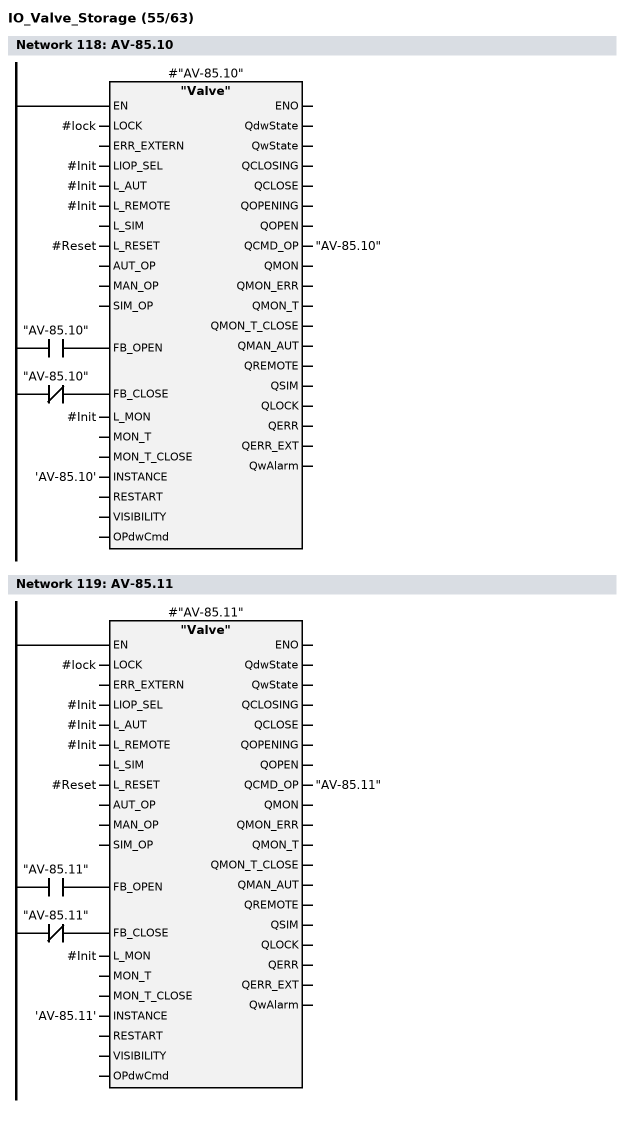
   RUNG wire#powerrail
      #"AV-85.10"(FB_OPEN := wire#w1, FB_CLOSE := wire#w2, LOCK := #lock, ERR_EXTERN :=, LIOP_SEL := #Init, L_AUT := #Init, L_REMOTE := #Init, L_SIM :=, L_RESET := #Reset, AUT_OP :=, MAN_OP :=, SIM_OP :=, L_MON := #Init, MON_T :=, MON_T_CLOSE :=, INSTANCE := 'AV-85.10', RESTART :=, VISIBILITY :=, OPdwCmd :=, QdwState =>, QwState =>, QCLOSING =>, QCLOSE =>, QOPENING =>, QOPEN =>, QCMD_OP => "AV-85.10", QMON =>, QMON_ERR =>, QMON_T =>, QMON_T_CLOSE =>, QMAN_AUT =>, QREMOTE =>, QSIM =>, QLOCK =>, QERR =>, QERR_EXT =>, QwAlarm =>)
   END_RUNG
   RUNG wire#powerrail
      Contact( "AV-85.10" )
   END_RUNG wire#w1
   RUNG wire#powerrail
      I_Contact( "AV-85.10" )
   END_RUNG wire#w2
   // the same network as SCL:
   #"AV-85.10"(LOCK := #lock,   // "Valve"
               LIOP_SEL := #Init,
               L_AUT := #Init,
               L_REMOTE := #Init,
               L_RESET := #Reset,
               FB_OPEN := "AV-85.10",
               FB_CLOSE := NOT "AV-85.10",
               L_MON := #Init,
               INSTANCE := 'AV-85.10',
               QCMD_OP => "AV-85.10");
END_REGION

REGION Network 119: AV-85.11
   RUNG wire#powerrail
      #"AV-85.11"(FB_OPEN := wire#w1, FB_CLOSE := wire#w2, LOCK := #lock, ERR_EXTERN :=, LIOP_SEL := #Init, L_AUT := #Init, L_REMOTE := #Init, L_SIM :=, L_RESET := #Reset, AUT_OP :=, MAN_OP :=, SIM_OP :=, L_MON := #Init, MON_T :=, MON_T_CLOSE :=, INSTANCE := 'AV-85.11', RESTART :=, VISIBILITY :=, OPdwCmd :=, QdwState =>, QwState =>, QCLOSING =>, QCLOSE =>, QOPENING =>, QOPEN =>, QCMD_OP => "AV-85.11", QMON =>, QMON_ERR =>, QMON_T =>, QMON_T_CLOSE =>, QMAN_AUT =>, QREMOTE =>, QSIM =>, QLOCK =>, QERR =>, QERR_EXT =>, QwAlarm =>)
   END_RUNG
   RUNG wire#powerrail
      Contact( "AV-85.11" )
   END_RUNG wire#w1
   RUNG wire#powerrail
      I_Contact( "AV-85.11" )
   END_RUNG wire#w2
   // the same network as SCL:
   #"AV-85.11"(LOCK := #lock,   // "Valve"
               LIOP_SEL := #Init,
               L_AUT := #Init,
               L_REMOTE := #Init,
               L_RESET := #Reset,
               FB_OPEN := "AV-85.11",
               FB_CLOSE := NOT "AV-85.11",
               L_MON := #Init,
               INSTANCE := 'AV-85.11',
               QCMD_OP => "AV-85.11");
END_REGION

REGION Network 120: AV-85.12
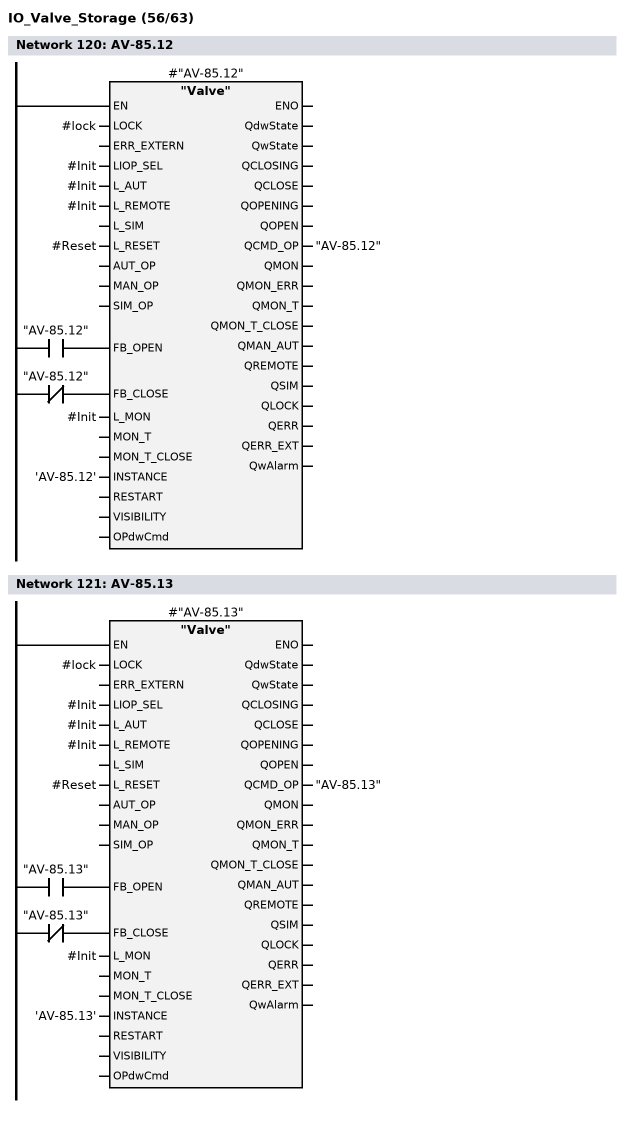
   RUNG wire#powerrail
      #"AV-85.12"(FB_OPEN := wire#w1, FB_CLOSE := wire#w2, LOCK := #lock, ERR_EXTERN :=, LIOP_SEL := #Init, L_AUT := #Init, L_REMOTE := #Init, L_SIM :=, L_RESET := #Reset, AUT_OP :=, MAN_OP :=, SIM_OP :=, L_MON := #Init, MON_T :=, MON_T_CLOSE :=, INSTANCE := 'AV-85.12', RESTART :=, VISIBILITY :=, OPdwCmd :=, QdwState =>, QwState =>, QCLOSING =>, QCLOSE =>, QOPENING =>, QOPEN =>, QCMD_OP => "AV-85.12", QMON =>, QMON_ERR =>, QMON_T =>, QMON_T_CLOSE =>, QMAN_AUT =>, QREMOTE =>, QSIM =>, QLOCK =>, QERR =>, QERR_EXT =>, QwAlarm =>)
   END_RUNG
   RUNG wire#powerrail
      Contact( "AV-85.12" )
   END_RUNG wire#w1
   RUNG wire#powerrail
      I_Contact( "AV-85.12" )
   END_RUNG wire#w2
   // the same network as SCL:
   #"AV-85.12"(LOCK := #lock,   // "Valve"
               LIOP_SEL := #Init,
               L_AUT := #Init,
               L_REMOTE := #Init,
               L_RESET := #Reset,
               FB_OPEN := "AV-85.12",
               FB_CLOSE := NOT "AV-85.12",
               L_MON := #Init,
               INSTANCE := 'AV-85.12',
               QCMD_OP => "AV-85.12");
END_REGION

REGION Network 121: AV-85.13
   RUNG wire#powerrail
      #"AV-85.13"(FB_OPEN := wire#w1, FB_CLOSE := wire#w2, LOCK := #lock, ERR_EXTERN :=, LIOP_SEL := #Init, L_AUT := #Init, L_REMOTE := #Init, L_SIM :=, L_RESET := #Reset, AUT_OP :=, MAN_OP :=, SIM_OP :=, L_MON := #Init, MON_T :=, MON_T_CLOSE :=, INSTANCE := 'AV-85.13', RESTART :=, VISIBILITY :=, OPdwCmd :=, QdwState =>, QwState =>, QCLOSING =>, QCLOSE =>, QOPENING =>, QOPEN =>, QCMD_OP => "AV-85.13", QMON =>, QMON_ERR =>, QMON_T =>, QMON_T_CLOSE =>, QMAN_AUT =>, QREMOTE =>, QSIM =>, QLOCK =>, QERR =>, QERR_EXT =>, QwAlarm =>)
   END_RUNG
   RUNG wire#powerrail
      Contact( "AV-85.13" )
   END_RUNG wire#w1
   RUNG wire#powerrail
      I_Contact( "AV-85.13" )
   END_RUNG wire#w2
   // the same network as SCL:
   #"AV-85.13"(LOCK := #lock,   // "Valve"
               LIOP_SEL := #Init,
               L_AUT := #Init,
               L_REMOTE := #Init,
               L_RESET := #Reset,
               FB_OPEN := "AV-85.13",
               FB_CLOSE := NOT "AV-85.13",
               L_MON := #Init,
               INSTANCE := 'AV-85.13',
               QCMD_OP => "AV-85.13");
END_REGION

REGION Network 122: AV-85.14
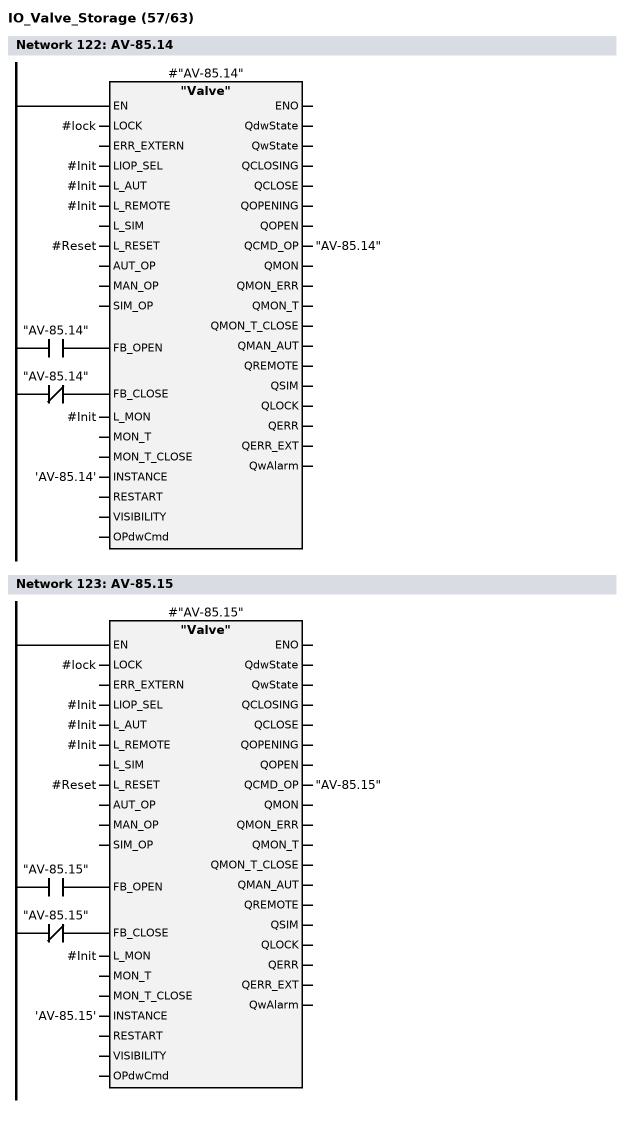
   RUNG wire#powerrail
      #"AV-85.14"(FB_OPEN := wire#w1, FB_CLOSE := wire#w2, LOCK := #lock, ERR_EXTERN :=, LIOP_SEL := #Init, L_AUT := #Init, L_REMOTE := #Init, L_SIM :=, L_RESET := #Reset, AUT_OP :=, MAN_OP :=, SIM_OP :=, L_MON := #Init, MON_T :=, MON_T_CLOSE :=, INSTANCE := 'AV-85.14', RESTART :=, VISIBILITY :=, OPdwCmd :=, QdwState =>, QwState =>, QCLOSING =>, QCLOSE =>, QOPENING =>, QOPEN =>, QCMD_OP => "AV-85.14", QMON =>, QMON_ERR =>, QMON_T =>, QMON_T_CLOSE =>, QMAN_AUT =>, QREMOTE =>, QSIM =>, QLOCK =>, QERR =>, QERR_EXT =>, QwAlarm =>)
   END_RUNG
   RUNG wire#powerrail
      Contact( "AV-85.14" )
   END_RUNG wire#w1
   RUNG wire#powerrail
      I_Contact( "AV-85.14" )
   END_RUNG wire#w2
   // the same network as SCL:
   #"AV-85.14"(LOCK := #lock,   // "Valve"
               LIOP_SEL := #Init,
               L_AUT := #Init,
               L_REMOTE := #Init,
               L_RESET := #Reset,
               FB_OPEN := "AV-85.14",
               FB_CLOSE := NOT "AV-85.14",
               L_MON := #Init,
               INSTANCE := 'AV-85.14',
               QCMD_OP => "AV-85.14");
END_REGION

REGION Network 123: AV-85.15
   RUNG wire#powerrail
      #"AV-85.15"(FB_OPEN := wire#w1, FB_CLOSE := wire#w2, LOCK := #lock, ERR_EXTERN :=, LIOP_SEL := #Init, L_AUT := #Init, L_REMOTE := #Init, L_SIM :=, L_RESET := #Reset, AUT_OP :=, MAN_OP :=, SIM_OP :=, L_MON := #Init, MON_T :=, MON_T_CLOSE :=, INSTANCE := 'AV-85.15', RESTART :=, VISIBILITY :=, OPdwCmd :=, QdwState =>, QwState =>, QCLOSING =>, QCLOSE =>, QOPENING =>, QOPEN =>, QCMD_OP => "AV-85.15", QMON =>, QMON_ERR =>, QMON_T =>, QMON_T_CLOSE =>, QMAN_AUT =>, QREMOTE =>, QSIM =>, QLOCK =>, QERR =>, QERR_EXT =>, QwAlarm =>)
   END_RUNG
   RUNG wire#powerrail
      Contact( "AV-85.15" )
   END_RUNG wire#w1
   RUNG wire#powerrail
      I_Contact( "AV-85.15" )
   END_RUNG wire#w2
   // the same network as SCL:
   #"AV-85.15"(LOCK := #lock,   // "Valve"
               LIOP_SEL := #Init,
               L_AUT := #Init,
               L_REMOTE := #Init,
               L_RESET := #Reset,
               FB_OPEN := "AV-85.15",
               FB_CLOSE := NOT "AV-85.15",
               L_MON := #Init,
               INSTANCE := 'AV-85.15',
               QCMD_OP => "AV-85.15");
END_REGION

REGION Network 124: AV-85.16
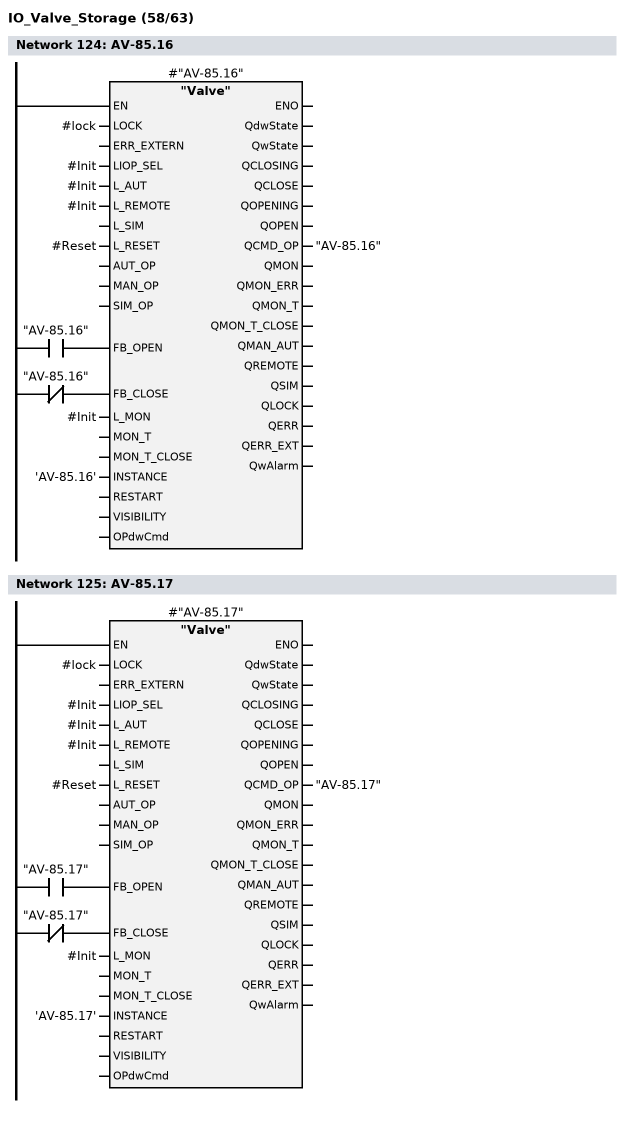
   RUNG wire#powerrail
      #"AV-85.16"(FB_OPEN := wire#w1, FB_CLOSE := wire#w2, LOCK := #lock, ERR_EXTERN :=, LIOP_SEL := #Init, L_AUT := #Init, L_REMOTE := #Init, L_SIM :=, L_RESET := #Reset, AUT_OP :=, MAN_OP :=, SIM_OP :=, L_MON := #Init, MON_T :=, MON_T_CLOSE :=, INSTANCE := 'AV-85.16', RESTART :=, VISIBILITY :=, OPdwCmd :=, QdwState =>, QwState =>, QCLOSING =>, QCLOSE =>, QOPENING =>, QOPEN =>, QCMD_OP => "AV-85.16", QMON =>, QMON_ERR =>, QMON_T =>, QMON_T_CLOSE =>, QMAN_AUT =>, QREMOTE =>, QSIM =>, QLOCK =>, QERR =>, QERR_EXT =>, QwAlarm =>)
   END_RUNG
   RUNG wire#powerrail
      Contact( "AV-85.16" )
   END_RUNG wire#w1
   RUNG wire#powerrail
      I_Contact( "AV-85.16" )
   END_RUNG wire#w2
   // the same network as SCL:
   #"AV-85.16"(LOCK := #lock,   // "Valve"
               LIOP_SEL := #Init,
               L_AUT := #Init,
               L_REMOTE := #Init,
               L_RESET := #Reset,
               FB_OPEN := "AV-85.16",
               FB_CLOSE := NOT "AV-85.16",
               L_MON := #Init,
               INSTANCE := 'AV-85.16',
               QCMD_OP => "AV-85.16");
END_REGION

REGION Network 125: AV-85.17
   RUNG wire#powerrail
      #"AV-85.17"(FB_OPEN := wire#w1, FB_CLOSE := wire#w2, LOCK := #lock, ERR_EXTERN :=, LIOP_SEL := #Init, L_AUT := #Init, L_REMOTE := #Init, L_SIM :=, L_RESET := #Reset, AUT_OP :=, MAN_OP :=, SIM_OP :=, L_MON := #Init, MON_T :=, MON_T_CLOSE :=, INSTANCE := 'AV-85.17', RESTART :=, VISIBILITY :=, OPdwCmd :=, QdwState =>, QwState =>, QCLOSING =>, QCLOSE =>, QOPENING =>, QOPEN =>, QCMD_OP => "AV-85.17", QMON =>, QMON_ERR =>, QMON_T =>, QMON_T_CLOSE =>, QMAN_AUT =>, QREMOTE =>, QSIM =>, QLOCK =>, QERR =>, QERR_EXT =>, QwAlarm =>)
   END_RUNG
   RUNG wire#powerrail
      Contact( "AV-85.17" )
   END_RUNG wire#w1
   RUNG wire#powerrail
      I_Contact( "AV-85.17" )
   END_RUNG wire#w2
   // the same network as SCL:
   #"AV-85.17"(LOCK := #lock,   // "Valve"
               LIOP_SEL := #Init,
               L_AUT := #Init,
               L_REMOTE := #Init,
               L_RESET := #Reset,
               FB_OPEN := "AV-85.17",
               FB_CLOSE := NOT "AV-85.17",
               L_MON := #Init,
               INSTANCE := 'AV-85.17',
               QCMD_OP => "AV-85.17");
END_REGION

REGION Network 126: AV-85.18
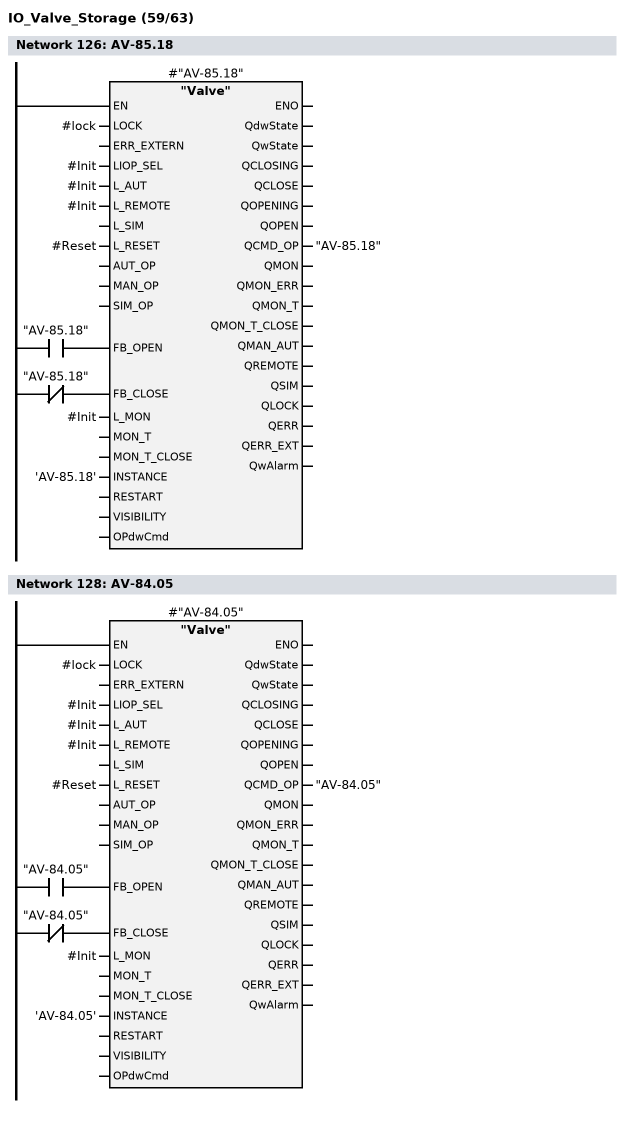
   RUNG wire#powerrail
      #"AV-85.18"(FB_OPEN := wire#w1, FB_CLOSE := wire#w2, LOCK := #lock, ERR_EXTERN :=, LIOP_SEL := #Init, L_AUT := #Init, L_REMOTE := #Init, L_SIM :=, L_RESET := #Reset, AUT_OP :=, MAN_OP :=, SIM_OP :=, L_MON := #Init, MON_T :=, MON_T_CLOSE :=, INSTANCE := 'AV-85.18', RESTART :=, VISIBILITY :=, OPdwCmd :=, QdwState =>, QwState =>, QCLOSING =>, QCLOSE =>, QOPENING =>, QOPEN =>, QCMD_OP => "AV-85.18", QMON =>, QMON_ERR =>, QMON_T =>, QMON_T_CLOSE =>, QMAN_AUT =>, QREMOTE =>, QSIM =>, QLOCK =>, QERR =>, QERR_EXT =>, QwAlarm =>)
   END_RUNG
   RUNG wire#powerrail
      Contact( "AV-85.18" )
   END_RUNG wire#w1
   RUNG wire#powerrail
      I_Contact( "AV-85.18" )
   END_RUNG wire#w2
   // the same network as SCL:
   #"AV-85.18"(LOCK := #lock,   // "Valve"
               LIOP_SEL := #Init,
               L_AUT := #Init,
               L_REMOTE := #Init,
               L_RESET := #Reset,
               FB_OPEN := "AV-85.18",
               FB_CLOSE := NOT "AV-85.18",
               L_MON := #Init,
               INSTANCE := 'AV-85.18',
               QCMD_OP => "AV-85.18");
END_REGION

REGION Network 128: AV-84.05
   RUNG wire#powerrail
      #"AV-84.05"(FB_OPEN := wire#w1, FB_CLOSE := wire#w2, LOCK := #lock, ERR_EXTERN :=, LIOP_SEL := #Init, L_AUT := #Init, L_REMOTE := #Init, L_SIM :=, L_RESET := #Reset, AUT_OP :=, MAN_OP :=, SIM_OP :=, L_MON := #Init, MON_T :=, MON_T_CLOSE :=, INSTANCE := 'AV-84.05', RESTART :=, VISIBILITY :=, OPdwCmd :=, QdwState =>, QwState =>, QCLOSING =>, QCLOSE =>, QOPENING =>, QOPEN =>, QCMD_OP => "AV-84.05", QMON =>, QMON_ERR =>, QMON_T =>, QMON_T_CLOSE =>, QMAN_AUT =>, QREMOTE =>, QSIM =>, QLOCK =>, QERR =>, QERR_EXT =>, QwAlarm =>)
   END_RUNG
   RUNG wire#powerrail
      Contact( "AV-84.05" )
   END_RUNG wire#w1
   RUNG wire#powerrail
      I_Contact( "AV-84.05" )
   END_RUNG wire#w2
   // the same network as SCL:
   #"AV-84.05"(LOCK := #lock,   // "Valve"
               LIOP_SEL := #Init,
               L_AUT := #Init,
               L_REMOTE := #Init,
               L_RESET := #Reset,
               FB_OPEN := "AV-84.05",
               FB_CLOSE := NOT "AV-84.05",
               L_MON := #Init,
               INSTANCE := 'AV-84.05',
               QCMD_OP => "AV-84.05");
END_REGION

REGION Network 129: AV-84.06
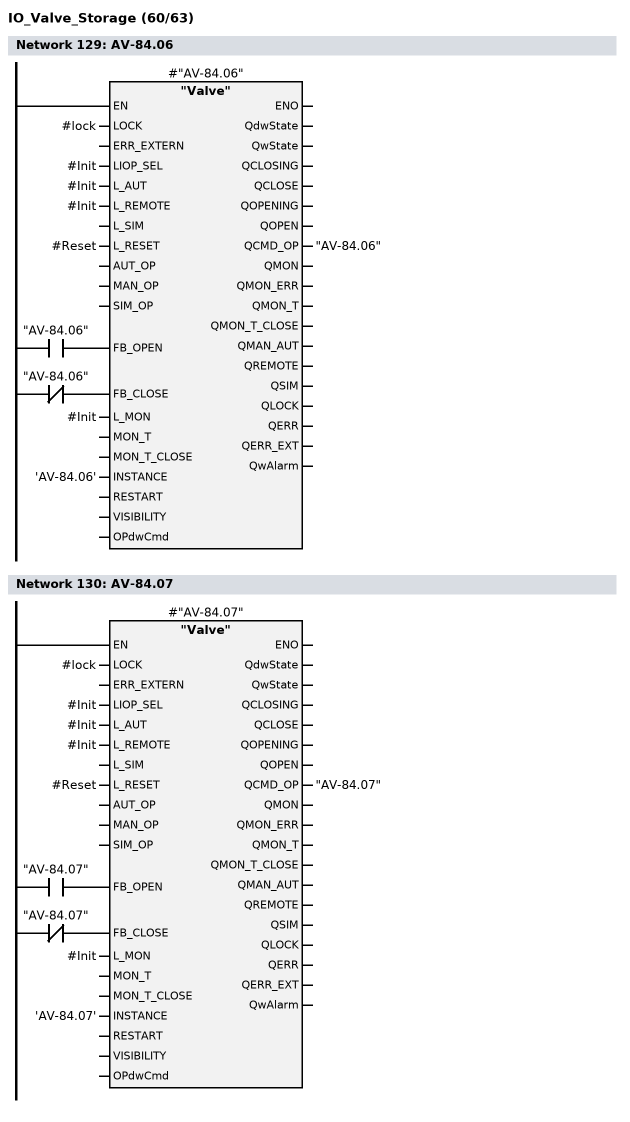
   RUNG wire#powerrail
      #"AV-84.06"(FB_OPEN := wire#w1, FB_CLOSE := wire#w2, LOCK := #lock, ERR_EXTERN :=, LIOP_SEL := #Init, L_AUT := #Init, L_REMOTE := #Init, L_SIM :=, L_RESET := #Reset, AUT_OP :=, MAN_OP :=, SIM_OP :=, L_MON := #Init, MON_T :=, MON_T_CLOSE :=, INSTANCE := 'AV-84.06', RESTART :=, VISIBILITY :=, OPdwCmd :=, QdwState =>, QwState =>, QCLOSING =>, QCLOSE =>, QOPENING =>, QOPEN =>, QCMD_OP => "AV-84.06", QMON =>, QMON_ERR =>, QMON_T =>, QMON_T_CLOSE =>, QMAN_AUT =>, QREMOTE =>, QSIM =>, QLOCK =>, QERR =>, QERR_EXT =>, QwAlarm =>)
   END_RUNG
   RUNG wire#powerrail
      Contact( "AV-84.06" )
   END_RUNG wire#w1
   RUNG wire#powerrail
      I_Contact( "AV-84.06" )
   END_RUNG wire#w2
   // the same network as SCL:
   #"AV-84.06"(LOCK := #lock,   // "Valve"
               LIOP_SEL := #Init,
               L_AUT := #Init,
               L_REMOTE := #Init,
               L_RESET := #Reset,
               FB_OPEN := "AV-84.06",
               FB_CLOSE := NOT "AV-84.06",
               L_MON := #Init,
               INSTANCE := 'AV-84.06',
               QCMD_OP => "AV-84.06");
END_REGION

REGION Network 130: AV-84.07
   RUNG wire#powerrail
      #"AV-84.07"(FB_OPEN := wire#w1, FB_CLOSE := wire#w2, LOCK := #lock, ERR_EXTERN :=, LIOP_SEL := #Init, L_AUT := #Init, L_REMOTE := #Init, L_SIM :=, L_RESET := #Reset, AUT_OP :=, MAN_OP :=, SIM_OP :=, L_MON := #Init, MON_T :=, MON_T_CLOSE :=, INSTANCE := 'AV-84.07', RESTART :=, VISIBILITY :=, OPdwCmd :=, QdwState =>, QwState =>, QCLOSING =>, QCLOSE =>, QOPENING =>, QOPEN =>, QCMD_OP => "AV-84.07", QMON =>, QMON_ERR =>, QMON_T =>, QMON_T_CLOSE =>, QMAN_AUT =>, QREMOTE =>, QSIM =>, QLOCK =>, QERR =>, QERR_EXT =>, QwAlarm =>)
   END_RUNG
   RUNG wire#powerrail
      Contact( "AV-84.07" )
   END_RUNG wire#w1
   RUNG wire#powerrail
      I_Contact( "AV-84.07" )
   END_RUNG wire#w2
   // the same network as SCL:
   #"AV-84.07"(LOCK := #lock,   // "Valve"
               LIOP_SEL := #Init,
               L_AUT := #Init,
               L_REMOTE := #Init,
               L_RESET := #Reset,
               FB_OPEN := "AV-84.07",
               FB_CLOSE := NOT "AV-84.07",
               L_MON := #Init,
               INSTANCE := 'AV-84.07',
               QCMD_OP => "AV-84.07");
END_REGION

REGION Network 131: AV-84.08
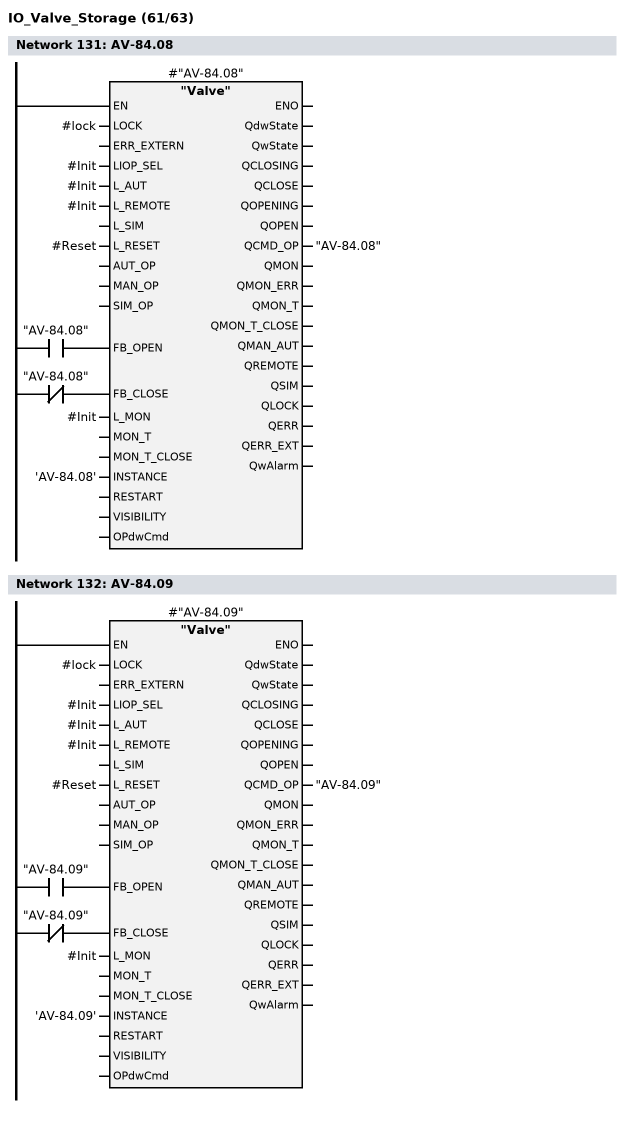
   RUNG wire#powerrail
      #"AV-84.08"(FB_OPEN := wire#w1, FB_CLOSE := wire#w2, LOCK := #lock, ERR_EXTERN :=, LIOP_SEL := #Init, L_AUT := #Init, L_REMOTE := #Init, L_SIM :=, L_RESET := #Reset, AUT_OP :=, MAN_OP :=, SIM_OP :=, L_MON := #Init, MON_T :=, MON_T_CLOSE :=, INSTANCE := 'AV-84.08', RESTART :=, VISIBILITY :=, OPdwCmd :=, QdwState =>, QwState =>, QCLOSING =>, QCLOSE =>, QOPENING =>, QOPEN =>, QCMD_OP => "AV-84.08", QMON =>, QMON_ERR =>, QMON_T =>, QMON_T_CLOSE =>, QMAN_AUT =>, QREMOTE =>, QSIM =>, QLOCK =>, QERR =>, QERR_EXT =>, QwAlarm =>)
   END_RUNG
   RUNG wire#powerrail
      Contact( "AV-84.08" )
   END_RUNG wire#w1
   RUNG wire#powerrail
      I_Contact( "AV-84.08" )
   END_RUNG wire#w2
   // the same network as SCL:
   #"AV-84.08"(LOCK := #lock,   // "Valve"
               LIOP_SEL := #Init,
               L_AUT := #Init,
               L_REMOTE := #Init,
               L_RESET := #Reset,
               FB_OPEN := "AV-84.08",
               FB_CLOSE := NOT "AV-84.08",
               L_MON := #Init,
               INSTANCE := 'AV-84.08',
               QCMD_OP => "AV-84.08");
END_REGION

REGION Network 132: AV-84.09
   RUNG wire#powerrail
      #"AV-84.09"(FB_OPEN := wire#w1, FB_CLOSE := wire#w2, LOCK := #lock, ERR_EXTERN :=, LIOP_SEL := #Init, L_AUT := #Init, L_REMOTE := #Init, L_SIM :=, L_RESET := #Reset, AUT_OP :=, MAN_OP :=, SIM_OP :=, L_MON := #Init, MON_T :=, MON_T_CLOSE :=, INSTANCE := 'AV-84.09', RESTART :=, VISIBILITY :=, OPdwCmd :=, QdwState =>, QwState =>, QCLOSING =>, QCLOSE =>, QOPENING =>, QOPEN =>, QCMD_OP => "AV-84.09", QMON =>, QMON_ERR =>, QMON_T =>, QMON_T_CLOSE =>, QMAN_AUT =>, QREMOTE =>, QSIM =>, QLOCK =>, QERR =>, QERR_EXT =>, QwAlarm =>)
   END_RUNG
   RUNG wire#powerrail
      Contact( "AV-84.09" )
   END_RUNG wire#w1
   RUNG wire#powerrail
      I_Contact( "AV-84.09" )
   END_RUNG wire#w2
   // the same network as SCL:
   #"AV-84.09"(LOCK := #lock,   // "Valve"
               LIOP_SEL := #Init,
               L_AUT := #Init,
               L_REMOTE := #Init,
               L_RESET := #Reset,
               FB_OPEN := "AV-84.09",
               FB_CLOSE := NOT "AV-84.09",
               L_MON := #Init,
               INSTANCE := 'AV-84.09',
               QCMD_OP => "AV-84.09");
END_REGION

REGION Network 133: AV-84.10
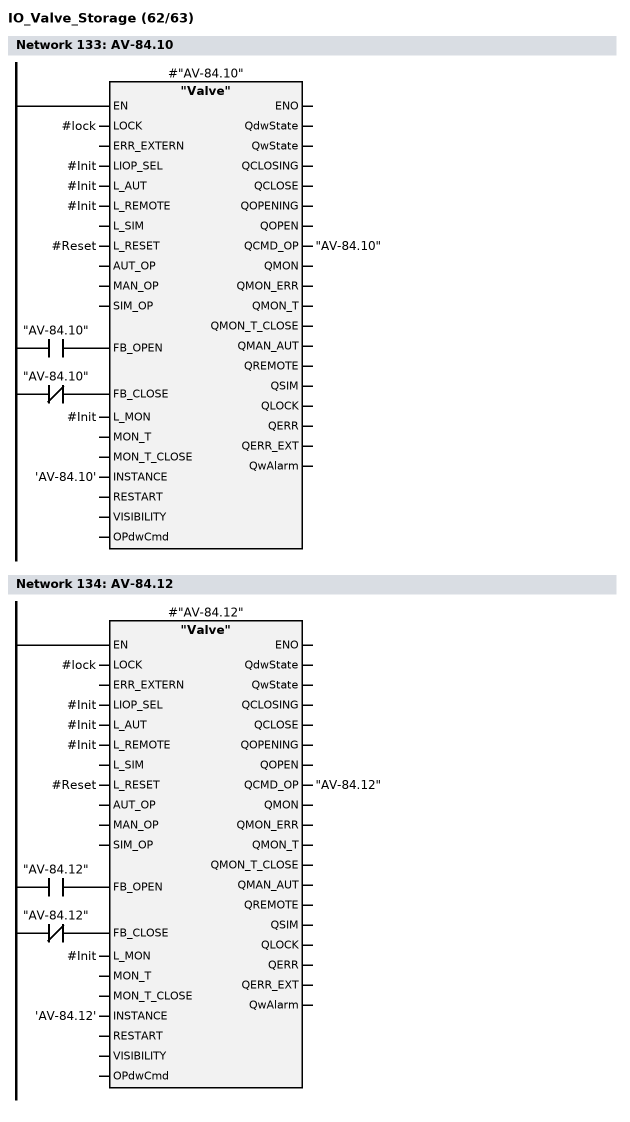
   RUNG wire#powerrail
      #"AV-84.10"(FB_OPEN := wire#w1, FB_CLOSE := wire#w2, LOCK := #lock, ERR_EXTERN :=, LIOP_SEL := #Init, L_AUT := #Init, L_REMOTE := #Init, L_SIM :=, L_RESET := #Reset, AUT_OP :=, MAN_OP :=, SIM_OP :=, L_MON := #Init, MON_T :=, MON_T_CLOSE :=, INSTANCE := 'AV-84.10', RESTART :=, VISIBILITY :=, OPdwCmd :=, QdwState =>, QwState =>, QCLOSING =>, QCLOSE =>, QOPENING =>, QOPEN =>, QCMD_OP => "AV-84.10", QMON =>, QMON_ERR =>, QMON_T =>, QMON_T_CLOSE =>, QMAN_AUT =>, QREMOTE =>, QSIM =>, QLOCK =>, QERR =>, QERR_EXT =>, QwAlarm =>)
   END_RUNG
   RUNG wire#powerrail
      Contact( "AV-84.10" )
   END_RUNG wire#w1
   RUNG wire#powerrail
      I_Contact( "AV-84.10" )
   END_RUNG wire#w2
   // the same network as SCL:
   #"AV-84.10"(LOCK := #lock,   // "Valve"
               LIOP_SEL := #Init,
               L_AUT := #Init,
               L_REMOTE := #Init,
               L_RESET := #Reset,
               FB_OPEN := "AV-84.10",
               FB_CLOSE := NOT "AV-84.10",
               L_MON := #Init,
               INSTANCE := 'AV-84.10',
               QCMD_OP => "AV-84.10");
END_REGION

REGION Network 134: AV-84.12
   RUNG wire#powerrail
      #"AV-84.12"(FB_OPEN := wire#w1, FB_CLOSE := wire#w2, LOCK := #lock, ERR_EXTERN :=, LIOP_SEL := #Init, L_AUT := #Init, L_REMOTE := #Init, L_SIM :=, L_RESET := #Reset, AUT_OP :=, MAN_OP :=, SIM_OP :=, L_MON := #Init, MON_T :=, MON_T_CLOSE :=, INSTANCE := 'AV-84.12', RESTART :=, VISIBILITY :=, OPdwCmd :=, QdwState =>, QwState =>, QCLOSING =>, QCLOSE =>, QOPENING =>, QOPEN =>, QCMD_OP => "AV-84.12", QMON =>, QMON_ERR =>, QMON_T =>, QMON_T_CLOSE =>, QMAN_AUT =>, QREMOTE =>, QSIM =>, QLOCK =>, QERR =>, QERR_EXT =>, QwAlarm =>)
   END_RUNG
   RUNG wire#powerrail
      Contact( "AV-84.12" )
   END_RUNG wire#w1
   RUNG wire#powerrail
      I_Contact( "AV-84.12" )
   END_RUNG wire#w2
   // the same network as SCL:
   #"AV-84.12"(LOCK := #lock,   // "Valve"
               LIOP_SEL := #Init,
               L_AUT := #Init,
               L_REMOTE := #Init,
               L_RESET := #Reset,
               FB_OPEN := "AV-84.12",
               FB_CLOSE := NOT "AV-84.12",
               L_MON := #Init,
               INSTANCE := 'AV-84.12',
               QCMD_OP => "AV-84.12");
END_REGION

REGION Network 135: AV-84.13
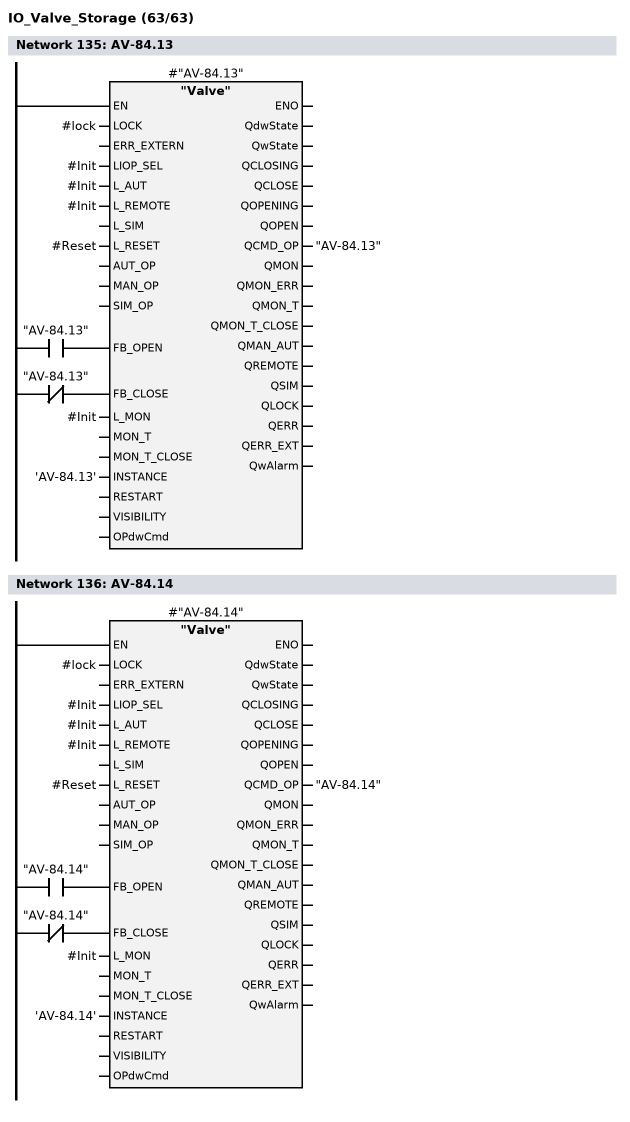
   RUNG wire#powerrail
      #"AV-84.13"(FB_OPEN := wire#w1, FB_CLOSE := wire#w2, LOCK := #lock, ERR_EXTERN :=, LIOP_SEL := #Init, L_AUT := #Init, L_REMOTE := #Init, L_SIM :=, L_RESET := #Reset, AUT_OP :=, MAN_OP :=, SIM_OP :=, L_MON := #Init, MON_T :=, MON_T_CLOSE :=, INSTANCE := 'AV-84.13', RESTART :=, VISIBILITY :=, OPdwCmd :=, QdwState =>, QwState =>, QCLOSING =>, QCLOSE =>, QOPENING =>, QOPEN =>, QCMD_OP => "AV-84.13", QMON =>, QMON_ERR =>, QMON_T =>, QMON_T_CLOSE =>, QMAN_AUT =>, QREMOTE =>, QSIM =>, QLOCK =>, QERR =>, QERR_EXT =>, QwAlarm =>)
   END_RUNG
   RUNG wire#powerrail
      Contact( "AV-84.13" )
   END_RUNG wire#w1
   RUNG wire#powerrail
      I_Contact( "AV-84.13" )
   END_RUNG wire#w2
   // the same network as SCL:
   #"AV-84.13"(LOCK := #lock,   // "Valve"
               LIOP_SEL := #Init,
               L_AUT := #Init,
               L_REMOTE := #Init,
               L_RESET := #Reset,
               FB_OPEN := "AV-84.13",
               FB_CLOSE := NOT "AV-84.13",
               L_MON := #Init,
               INSTANCE := 'AV-84.13',
               QCMD_OP => "AV-84.13");
END_REGION

REGION Network 136: AV-84.14
   RUNG wire#powerrail
      #"AV-84.14"(FB_OPEN := wire#w1, FB_CLOSE := wire#w2, LOCK := #lock, ERR_EXTERN :=, LIOP_SEL := #Init, L_AUT := #Init, L_REMOTE := #Init, L_SIM :=, L_RESET := #Reset, AUT_OP :=, MAN_OP :=, SIM_OP :=, L_MON := #Init, MON_T :=, MON_T_CLOSE :=, INSTANCE := 'AV-84.14', RESTART :=, VISIBILITY :=, OPdwCmd :=, QdwState =>, QwState =>, QCLOSING =>, QCLOSE =>, QOPENING =>, QOPEN =>, QCMD_OP => "AV-84.14", QMON =>, QMON_ERR =>, QMON_T =>, QMON_T_CLOSE =>, QMAN_AUT =>, QREMOTE =>, QSIM =>, QLOCK =>, QERR =>, QERR_EXT =>, QwAlarm =>)
   END_RUNG
   RUNG wire#powerrail
      Contact( "AV-84.14" )
   END_RUNG wire#w1
   RUNG wire#powerrail
      I_Contact( "AV-84.14" )
   END_RUNG wire#w2
   // the same network as SCL:
   #"AV-84.14"(LOCK := #lock,   // "Valve"
               LIOP_SEL := #Init,
               L_AUT := #Init,
               L_REMOTE := #Init,
               L_RESET := #Reset,
               FB_OPEN := "AV-84.14",
               FB_CLOSE := NOT "AV-84.14",
               L_MON := #Init,
               INSTANCE := 'AV-84.14',
               QCMD_OP => "AV-84.14");
END_REGION
END_FUNCTION_BLOCK

FUNCTION_BLOCK "IO_Digital_Storage"   // FB22, LAD
{ S7_Optimized_Access := 'TRUE' }
VERSION : 0.1
// stored: AutoNumber false, IsIECCheckEnabled false, IsRetainMemResEnabled false, MemoryReserve 100, SetENOAutomatically false, UDAEnableTagReadback false
   VAR_INPUT
      lock : Bool;
      init : Bool;
      Reset : Bool;
   END_VAR
   VAR
      "FS-23.01" : "Digital";
      "FS-24.01" { S7_SetPoint := 'True'} : "Digital";
      "FS-34.01" { S7_SetPoint := 'True'} : "Digital";
      "FS-35.01" { S7_SetPoint := 'True'} : "Digital";
   END_VAR
BEGIN

REGION Network 1: FS-23.01
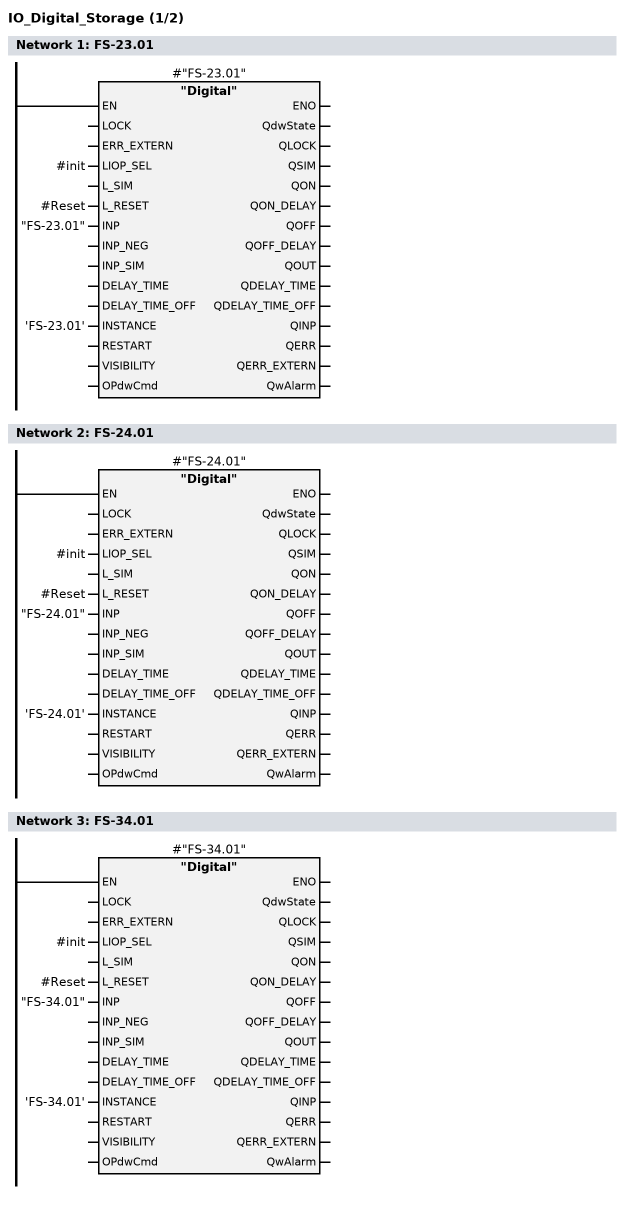
   RUNG wire#powerrail
      #"FS-23.01"(LOCK :=, ERR_EXTERN :=, LIOP_SEL := #init, L_SIM :=, L_RESET := #Reset, INP := "FS-23.01", INP_NEG :=, INP_SIM :=, DELAY_TIME :=, DELAY_TIME_OFF :=, INSTANCE := 'FS-23.01', RESTART :=, VISIBILITY :=, OPdwCmd :=, QdwState =>, QLOCK =>, QSIM =>, QON =>, QON_DELAY =>, QOFF =>, QOFF_DELAY =>, QOUT =>, QDELAY_TIME =>, QDELAY_TIME_OFF =>, QINP =>, QERR =>, QERR_EXTERN =>, QwAlarm =>)
   END_RUNG
   // the same network as SCL:
   #"FS-23.01"(LIOP_SEL := #init, L_RESET := #Reset, INP := "FS-23.01", INSTANCE := 'FS-23.01');   // "Digital"
END_REGION

REGION Network 2: FS-24.01
   RUNG wire#powerrail
      #"FS-24.01"(LOCK :=, ERR_EXTERN :=, LIOP_SEL := #init, L_SIM :=, L_RESET := #Reset, INP := "FS-24.01", INP_NEG :=, INP_SIM :=, DELAY_TIME :=, DELAY_TIME_OFF :=, INSTANCE := 'FS-24.01', RESTART :=, VISIBILITY :=, OPdwCmd :=, QdwState =>, QLOCK =>, QSIM =>, QON =>, QON_DELAY =>, QOFF =>, QOFF_DELAY =>, QOUT =>, QDELAY_TIME =>, QDELAY_TIME_OFF =>, QINP =>, QERR =>, QERR_EXTERN =>, QwAlarm =>)
   END_RUNG
   // the same network as SCL:
   #"FS-24.01"(LIOP_SEL := #init, L_RESET := #Reset, INP := "FS-24.01", INSTANCE := 'FS-24.01');   // "Digital"
END_REGION

REGION Network 3: FS-34.01
   RUNG wire#powerrail
      #"FS-34.01"(LOCK :=, ERR_EXTERN :=, LIOP_SEL := #init, L_SIM :=, L_RESET := #Reset, INP := "FS-34.01", INP_NEG :=, INP_SIM :=, DELAY_TIME :=, DELAY_TIME_OFF :=, INSTANCE := 'FS-34.01', RESTART :=, VISIBILITY :=, OPdwCmd :=, QdwState =>, QLOCK =>, QSIM =>, QON =>, QON_DELAY =>, QOFF =>, QOFF_DELAY =>, QOUT =>, QDELAY_TIME =>, QDELAY_TIME_OFF =>, QINP =>, QERR =>, QERR_EXTERN =>, QwAlarm =>)
   END_RUNG
   // the same network as SCL:
   #"FS-34.01"(LIOP_SEL := #init, L_RESET := #Reset, INP := "FS-34.01", INSTANCE := 'FS-34.01');   // "Digital"
END_REGION

REGION Network 4: FS-35.01
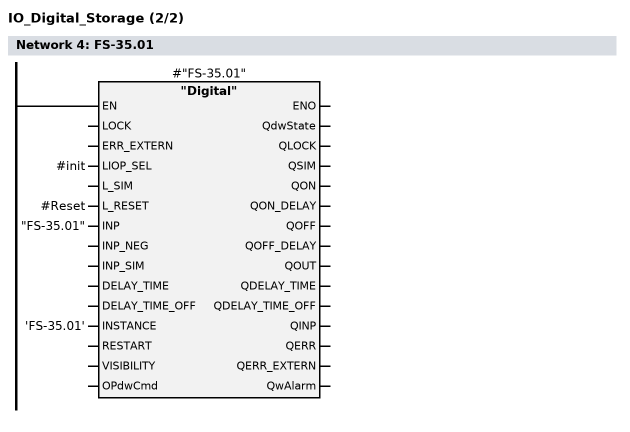
   RUNG wire#powerrail
      #"FS-35.01"(LOCK :=, ERR_EXTERN :=, LIOP_SEL := #init, L_SIM :=, L_RESET := #Reset, INP := "FS-35.01", INP_NEG :=, INP_SIM :=, DELAY_TIME :=, DELAY_TIME_OFF :=, INSTANCE := 'FS-35.01', RESTART :=, VISIBILITY :=, OPdwCmd :=, QdwState =>, QLOCK =>, QSIM =>, QON =>, QON_DELAY =>, QOFF =>, QOFF_DELAY =>, QOUT =>, QDELAY_TIME =>, QDELAY_TIME_OFF =>, QINP =>, QERR =>, QERR_EXTERN =>, QwAlarm =>)
   END_RUNG
   // the same network as SCL:
   #"FS-35.01"(LIOP_SEL := #init, L_RESET := #Reset, INP := "FS-35.01", INSTANCE := 'FS-35.01');   // "Digital"
END_REGION
END_FUNCTION_BLOCK

FUNCTION_BLOCK "Storage_Tank_Single_Inload"   // FB21, LAD
{ S7_Optimized_Access := 'FALSE' }
VERSION : 0.1
// stored: AutoNumber true, IsIECCheckEnabled false, SetENOAutomatically false, UDAEnableTagReadback false
   VAR_INPUT
      Level_Bypass : Bool;
      Single_CIP_Cmd : Bool;
      IN_FBAV_Load : Bool;
      IN_FBAV_Transfer : Bool;
      IN_FBP_Transfer : Bool;
      IN_FBP_Transfer_Speed : Real;
      IN_FBP_CIP : Bool;
      IN_FBAV_CIP_Sup : Bool;
      IN_FBAV_CIP_Tank : Bool;
      IN_FBAV_CIP_Line : Bool;
      IN_LT01 : Real;
      IN_FS : Bool;
      CIP_Req_OK : Bool;
      CIP_ON_Progress : Bool;
      CIP_Supply_ON : Bool;
      CIP_Complete : Bool;
      CIPPulse : Bool;
      Filler_Product_Req : Bool;
      Filler_CIP_Req : Bool;
      Loading_Busy : Bool;
      Transfer_Busy : Bool;
   END_VAR
   VAR_OUTPUT
      Out_AV_Load : Bool;
      Out_AV_Transfer : Bool;
      Out_P_Transfer : Bool;
      Out_P_TF_Speed : Real;
      Out_P_CIP : Bool;
      Out_AV_CIP_Line : Bool;
      Out_AV_CIP_Tank : Bool;
      Out_AV_CIP_Filling : Bool;
      CIP_Tank_Req : Bool;
      CIP_Line_Req : Bool;
      CIP_LineOK : Bool;
   END_VAR
   VAR DB_SPECIFIC
      Cmd : Struct
         Inload_Select_Tank : Bool;
         Inload : Bool;   // Start Loading
         Tank_CIP_Req : Bool;
         Line_CIP_Req : Bool;
         Tank_Filling_CIP_Req : Bool;
         CIP_Filling_En : Bool;
         CIP_Line_Req_OK : Bool;
         CIP_Supply_ON : Bool;
         CIP_ON_Progress : Bool;
         Flushing : Bool;   // Water Flushing
         RaadyForTF : Bool;   // Tank Ready for Blending
         Flush_Select : Byte;
         Drain_In : Bool;
         Drain_Transfer : Bool;
      END_STRUCT;
      Param : Struct
         SP_Level_LL : Real := 10.0;
         SP_Level_ML : Real := 80.0;
         SP_Level_HL : Real := 100.0;
         SupplyPump_SP_Speed : Real := 80.0;
         L_Hi_Lim : Real := 100.0;
         L_Lo_Lim : Real := 0.0;
         L_Hys : Real := 2.0;
         FlushingTime : DInt := 10000;
         CIP_Trf_SP_Speed : Real := 80.0;
         CIP_Ret_ON_SP : Real := 10.0;
         CIP_Ret_OFF_SP : Real;
         Transfer_P_Speed : Real := 60.0;
         Drain_Inload_SP : DInt := 10;
         Drain_Transfer_SP : DInt := 10;
      END_STRUCT;
      State : Struct   // Tank in loading state
         Tank_inloading : Bool;
         Tank_inCIP : Bool;
         Tank_Filling_inCIP : Bool;
         Line_inCIP : Bool;
         FIlling_inCIP : Bool;
         Flushing : Bool;
         Tank_LL : Bool;
         Tank_ML : Bool;
         Tank_HL : Bool;
         Inload_Enable : Bool;
         Tank_CIP_Enable : Bool;
         Line_CIP_Enable : Bool;
         Tank_Filling_CIP_Enable : Bool;
         Flushing_Enable : Bool;
         Flush_selected : Byte;
         CIP_Request_OK : Bool;
         CIP_ReturnON : Bool;
         Ready_For_Transfer_EN : Bool;   // Tank Ready for Transfer to Blending
         Ready_For_Transfer : Bool;   // Tank Ready for Transfer to Blending
         HWT_Status : Int;
         Transfer_to_Filling : Bool;
         "Line_AV4&AV5" : Bool;
         "Line_AV1&AV2" : Bool;
         "Line_AV7&AV8" : Bool;
         "Line_AV10&AV11" : Bool;
         "Line_AV5&AV6" : Bool;
         CIP_Line1_ON : Bool;
         CIP_Line2_ON : Bool;
         CIP_Line3_ON : Bool;
         CIP_Line4_ON : Bool;
         Drain_Inload : Bool;
         Drain_Transfer : Bool;
      END_STRUCT;
      alwaysON : Bool;
      L_Hys_Abs : Real;
      Hys_Level_HL : Real;
      Hys_Level_ML : Real;
      Hys_Level_LL : Real;
      Drain_Inload_MSec : DInt;
      Drain_Inload_Count : IEC_DCOUNTER;
      Drain_Inload_Act { S7_SetPoint := 'True'} : DInt;
      Drain_Transfer_MSec : DInt;
      Drain_Transfer_Count : IEC_DCOUNTER;
      Drain_Transfer_Act : DInt;
      r : Struct
         PosE1 : Bool;
         PosE2 : Bool;
         PosE3 : Bool;
         PosE4 : Bool;
         PosE5 : Bool;
         PosE6 : Bool;
         PosE7 : Bool;
         PosE8 : Bool;
         PosE9 : Bool;
         PosE10 : Bool;
         PosE11 : Bool;
         PosE12 : Bool;
         PosE13 : Bool;
         PosE14 : Bool;
         PosE15 : Bool;
         PosE16 : Bool;
         PosE17 : Bool;
         PosE18 : Bool;
         PosE19 : Bool;
         PosE20 : Bool;
         PosE21 : Bool;
         PosE22 : Bool;
         PosE23 : Bool;
         PosE24 : Bool;
         PosE25 : Bool;
         PosE26 : Bool;
         PosE27 : Bool;
         PosE28 : Bool;
         PosE29 : Bool;
         PosE30 : Bool;
         PosE31 : Bool;
         PosE32 : Bool;
      END_STRUCT;
      Actuator : Struct
         AV_Outlet : Bool;
         AV_Load : Bool;
         AV_Transfer : Bool;
         CIP_Line_Pump : Bool;
         CIP_Tank_Pump : Bool;
         TransferPump : Bool;
         FlushPump : Bool;
         CV_Steam : Bool;
         Pump : Bool;
      END_STRUCT;
      SPumpTim { S7_SetPoint := 'True'} : TON_TIME;
      SAV_CIPLine { S7_SetPoint := 'True'} : TON_TIME;
      SAV_CIPTANK { S7_SetPoint := 'True'} : TON_TIME;
      SAV_CIPFILLING { S7_SetPoint := 'True'} : TON_TIME;
      AVinloadTim { S7_SetPoint := 'True'} : TON_TIME;
      AVOutletTim { S7_SetPoint := 'True'} : TON_TIME;
      Drain_In_Tim { S7_SetPoint := 'True'} : TON_TIME;
      Drain_Out_Tim { S7_SetPoint := 'True'} : TON_TIME;
      "Pump Off Tim" { S7_SetPoint := 'True'} : TON_TIME;
      "Loading_Busy Tim" { S7_SetPoint := 'True'} : TON_TIME;
   END_VAR
   VAR_TEMP   // added for the SCL form of the ladder/FBD networks
      _w1 : Bool;
      _w2 : Bool;
      _w3 : Bool;
      _w4 : Bool;
      _w5 : Bool;
      _w6 : Bool;
      _w7 : Bool;
   END_VAR
BEGIN

REGION Network 1: Always ON
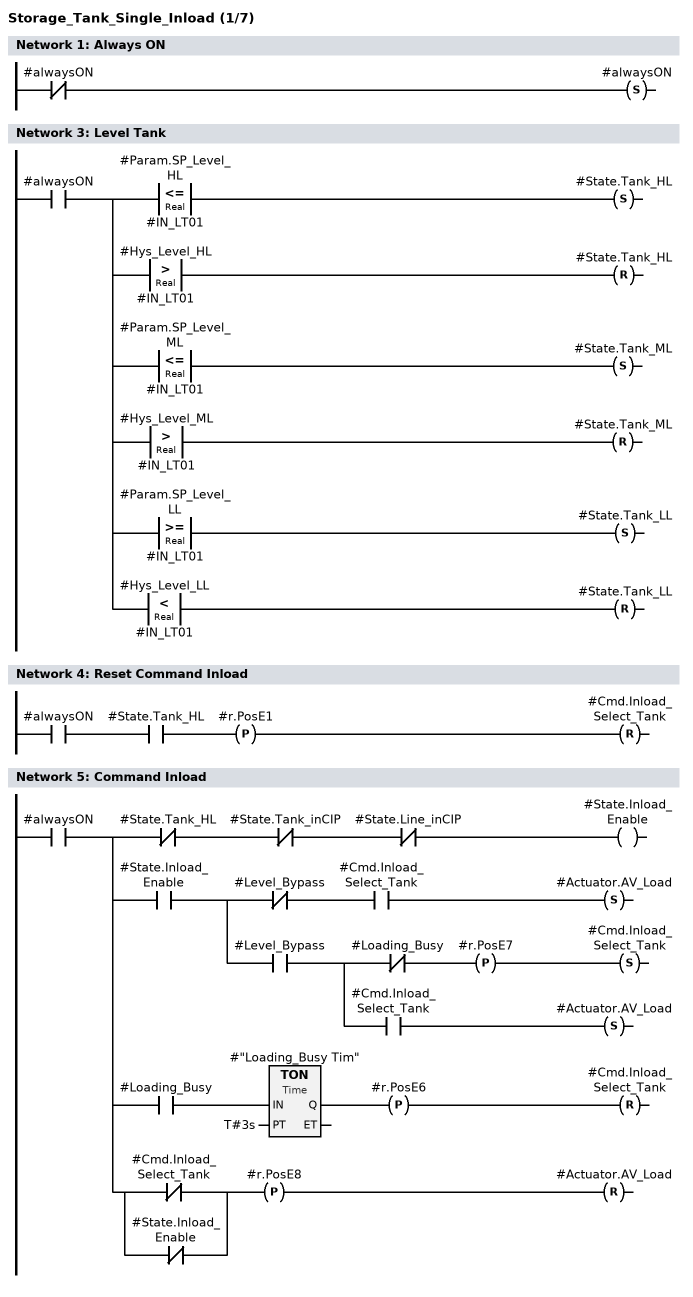
   RUNG wire#powerrail
      I_Contact( #alwaysON )
      S_Coil( #alwaysON )
   END_RUNG
   // the same network as SCL:
   IF NOT #alwaysON THEN #alwaysON := TRUE; END_IF;
END_REGION

NETWORK
TITLE = Hys Calculation
//Level Hys Absolute
      L     #Param.L_Hi_Lim;
      L     #Param.L_Lo_Lim;
      -R;
      L     100.0;
      /R;
      L     #Param.L_Hys;
      *R;
      T     #L_Hys_Abs;
//Tank High Level
      L     #Param.SP_Level_HL;
      L     #L_Hys_Abs;
      -R;
      T     #Hys_Level_HL;
//Tank Mid Level
      L     #Param.SP_Level_ML;
      L     #L_Hys_Abs;
      -R;
      T     #Hys_Level_ML;
//Tank Low Level
      L     #Param.SP_Level_LL;
      L     #L_Hys_Abs;
      +R;
      T     #Hys_Level_LL;


REGION Network 3: Level Tank
   RUNG wire#powerrail
      Contact( #alwaysON )
      wire#w1
      { S7_Templates := "SrcType := Real" } LE_Contact(in1 := #Param.SP_Level_HL, in2 := #IN_LT01)
      S_Coil( #State.Tank_HL )
   END_RUNG
   RUNG wire#w1
      { S7_Templates := "SrcType := Real" } GT_Contact(in1 := #Hys_Level_HL, in2 := #IN_LT01)
      R_Coil( #State.Tank_HL )
   END_RUNG
   RUNG wire#w1
      { S7_Templates := "SrcType := Real" } LE_Contact(in1 := #Param.SP_Level_ML, in2 := #IN_LT01)
      S_Coil( #State.Tank_ML )
   END_RUNG
   RUNG wire#w1
      { S7_Templates := "SrcType := Real" } GT_Contact(in1 := #Hys_Level_ML, in2 := #IN_LT01)
      R_Coil( #State.Tank_ML )
   END_RUNG
   RUNG wire#w1
      { S7_Templates := "SrcType := Real" } GE_Contact(in1 := #Param.SP_Level_LL, in2 := #IN_LT01)
      S_Coil( #State.Tank_LL )
   END_RUNG
   RUNG wire#w1
      { S7_Templates := "SrcType := Real" } LT_Contact(in1 := #Hys_Level_LL, in2 := #IN_LT01)
      R_Coil( #State.Tank_LL )
   END_RUNG
   // the same network as SCL:
   IF #alwaysON AND (#Param.SP_Level_HL <= #IN_LT01) THEN #State.Tank_HL := TRUE; END_IF;
   IF #alwaysON AND (#Hys_Level_HL > #IN_LT01) THEN #State.Tank_HL := FALSE; END_IF;
   IF #alwaysON AND (#Param.SP_Level_ML <= #IN_LT01) THEN #State.Tank_ML := TRUE; END_IF;
   IF #alwaysON AND (#Hys_Level_ML > #IN_LT01) THEN #State.Tank_ML := FALSE; END_IF;
   IF #alwaysON AND (#Param.SP_Level_LL >= #IN_LT01) THEN #State.Tank_LL := TRUE; END_IF;
   IF #alwaysON AND (#Hys_Level_LL < #IN_LT01) THEN #State.Tank_LL := FALSE; END_IF;
END_REGION

REGION Network 4: Reset Command Inload
   RUNG wire#powerrail
      Contact( #alwaysON )
      Contact( #State.Tank_HL )
      P_Trig( #r.PosE1 )
      R_Coil( #Cmd.Inload_Select_Tank )
   END_RUNG
   // the same network as SCL:
   #_w1 := #alwaysON AND #State.Tank_HL;
   #_w2 := #_w1 AND NOT #r.PosE1;   // rising edge
   #r.PosE1 := #_w1;
   IF #_w2 THEN #Cmd.Inload_Select_Tank := FALSE; END_IF;
END_REGION

REGION Network 5: Command Inload
   RUNG wire#powerrail
      Contact( #alwaysON )
      wire#w1
      I_Contact( #State.Tank_HL )
      I_Contact( #State.Tank_inCIP )
      I_Contact( #State.Line_inCIP )
      Coil( #State.Inload_Enable )
   END_RUNG
   RUNG wire#w1
      Contact( #State.Inload_Enable )
      wire#w2
      I_Contact( #Level_Bypass )
      Contact( #Cmd.Inload_Select_Tank )
      S_Coil( #Actuator.AV_Load )
   END_RUNG
   RUNG wire#w2
      Contact( #Level_Bypass )
      wire#w3
      I_Contact( #Loading_Busy )
      P_Trig( #r.PosE7 )
      S_Coil( #Cmd.Inload_Select_Tank )
   END_RUNG
   RUNG wire#w3
      Contact( #Cmd.Inload_Select_Tank )
      S_Coil( #Actuator.AV_Load )
   END_RUNG
   RUNG wire#w1
      Contact( #Loading_Busy )
      { S7_Templates := "time_type := Time" } #"Loading_Busy Tim".TON(pt := T#3s, et =>)
      P_Trig( #r.PosE6 )
      R_Coil( #Cmd.Inload_Select_Tank )
   END_RUNG
   RUNG wire#w1
      I_Contact( #Cmd.Inload_Select_Tank )
      wire#w4
      P_Trig( #r.PosE8 )
      R_Coil( #Actuator.AV_Load )
   END_RUNG
   RUNG wire#w1
      I_Contact( #State.Inload_Enable )
   END_RUNG wire#w4
   // the same network as SCL:
   #State.Inload_Enable := #alwaysON AND NOT #State.Tank_HL AND NOT #State.Tank_inCIP AND NOT #State.Line_inCIP;
   #_w1 := #alwaysON AND #State.Inload_Enable;
   IF #_w1 AND NOT #Level_Bypass AND #Cmd.Inload_Select_Tank THEN #Actuator.AV_Load := TRUE; END_IF;
   #_w2 := #_w1 AND #Level_Bypass;
   #_w3 := #_w2 AND NOT #Loading_Busy;
   #_w4 := #_w3 AND NOT #r.PosE7;   // rising edge
   #r.PosE7 := #_w3;
   IF #_w4 THEN #Cmd.Inload_Select_Tank := TRUE; END_IF;
   IF #_w2 AND #Cmd.Inload_Select_Tank THEN #Actuator.AV_Load := TRUE; END_IF;
   #"Loading_Busy Tim"(IN := #alwaysON AND #Loading_Busy, PT := T#3s);   // TON
   #_w5 := #"Loading_Busy Tim".Q AND NOT #r.PosE6;   // rising edge
   #r.PosE6 := #"Loading_Busy Tim".Q;
   IF #_w5 THEN #Cmd.Inload_Select_Tank := FALSE; END_IF;
   #_w6 := #alwaysON AND (NOT #Cmd.Inload_Select_Tank OR NOT #State.Inload_Enable);
   #_w7 := #_w6 AND NOT #r.PosE8;   // rising edge
   #r.PosE8 := #_w6;
   IF #_w7 THEN #Actuator.AV_Load := FALSE; END_IF;
END_REGION

REGION Network 6: Drain Inload
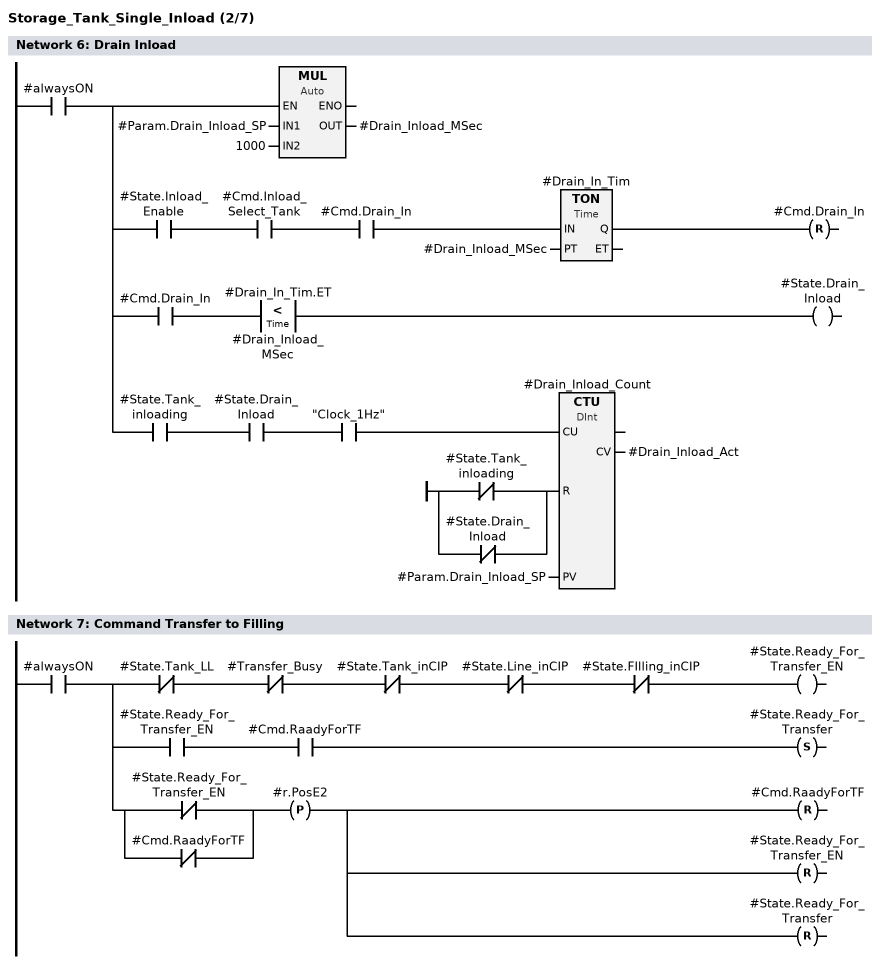
   RUNG wire#powerrail
      Contact( #alwaysON )
      wire#w1
      Mul(in1 := #Param.Drain_Inload_SP, in2 := 1000, out => #Drain_Inload_MSec)
   END_RUNG
   RUNG wire#w1
      Contact( #State.Inload_Enable )
      Contact( #Cmd.Inload_Select_Tank )
      Contact( #Cmd.Drain_In )
      { S7_Templates := "time_type := Time" } #Drain_In_Tim.TON(pt := #Drain_Inload_MSec, et =>)
      R_Coil( #Cmd.Drain_In )
   END_RUNG
   RUNG wire#w1
      Contact( #Cmd.Drain_In )
      { S7_Templates := "SrcType := Time" } LT_Contact(in1 := #Drain_In_Tim.ET, in2 := #Drain_Inload_MSec)
      Coil( #State.Drain_Inload )
   END_RUNG
   RUNG wire#w1
      Contact( #State.Tank_inloading )
      Contact( #State.Drain_Inload )
      Contact( "Clock_1Hz" )
      { S7_Templates := "value_type := DInt" } #Drain_Inload_Count.CTU(r := wire#w2, pv := #Param.Drain_Inload_SP, cv => #Drain_Inload_Act)
   END_RUNG
   RUNG wire#powerrail
      I_Contact( #State.Tank_inloading )
   END_RUNG wire#w2
   RUNG wire#powerrail
      I_Contact( #State.Drain_Inload )
   END_RUNG wire#w2
   // the same network as SCL:
   IF #alwaysON THEN #Drain_Inload_MSec := #Param.Drain_Inload_SP * 1000; END_IF;
   #Drain_In_Tim(IN := #alwaysON AND #State.Inload_Enable AND #Cmd.Inload_Select_Tank AND #Cmd.Drain_In,   // TON
                 PT := #Drain_Inload_MSec);
   IF #Drain_In_Tim.Q THEN #Cmd.Drain_In := FALSE; END_IF;
   #State.Drain_Inload := #alwaysON AND #Cmd.Drain_In AND (#Drain_In_Tim.ET < #Drain_Inload_MSec);
   #Drain_Inload_Count.CTU(CU := #alwaysON AND #State.Tank_inloading AND #State.Drain_Inload AND "Clock_1Hz",
                           R := NOT #State.Tank_inloading OR NOT #State.Drain_Inload,
                           PV := #Param.Drain_Inload_SP,
                           CV => #Drain_Inload_Act);
END_REGION

REGION Network 7: Command Transfer to Filling
   RUNG wire#powerrail
      Contact( #alwaysON )
      wire#w1
      I_Contact( #State.Tank_LL )
      I_Contact( #Transfer_Busy )
      I_Contact( #State.Tank_inCIP )
      I_Contact( #State.Line_inCIP )
      I_Contact( #State.FIlling_inCIP )
      Coil( #State.Ready_For_Transfer_EN )
   END_RUNG
   RUNG wire#w1
      Contact( #State.Ready_For_Transfer_EN )
      Contact( #Cmd.RaadyForTF )
      S_Coil( #State.Ready_For_Transfer )
   END_RUNG
   RUNG wire#w1
      I_Contact( #State.Ready_For_Transfer_EN )
      wire#w2
      P_Trig( #r.PosE2 )
      wire#w3
      R_Coil( #Cmd.RaadyForTF )
   END_RUNG
   RUNG wire#w1
      I_Contact( #Cmd.RaadyForTF )
   END_RUNG wire#w2
   RUNG wire#w3
      R_Coil( #State.Ready_For_Transfer_EN )
   END_RUNG
   RUNG wire#w3
      R_Coil( #State.Ready_For_Transfer )
   END_RUNG
   // the same network as SCL:
   #State.Ready_For_Transfer_EN := #alwaysON AND NOT #State.Tank_LL AND NOT #Transfer_Busy AND NOT #State.Tank_inCIP AND NOT #State.Line_inCIP AND NOT #State.FIlling_inCIP;
   IF #alwaysON AND #State.Ready_For_Transfer_EN AND #Cmd.RaadyForTF THEN
       #State.Ready_For_Transfer := TRUE;
   END_IF;
   #_w1 := #alwaysON AND (NOT #State.Ready_For_Transfer_EN OR NOT #Cmd.RaadyForTF);
   #_w2 := #_w1 AND NOT #r.PosE2;   // rising edge
   #r.PosE2 := #_w1;
   IF #_w2 THEN
       #Cmd.RaadyForTF := FALSE;
       #State.Ready_For_Transfer_EN := FALSE;
       #State.Ready_For_Transfer := FALSE;
   END_IF;
END_REGION

REGION Network 8: Drain Transfer
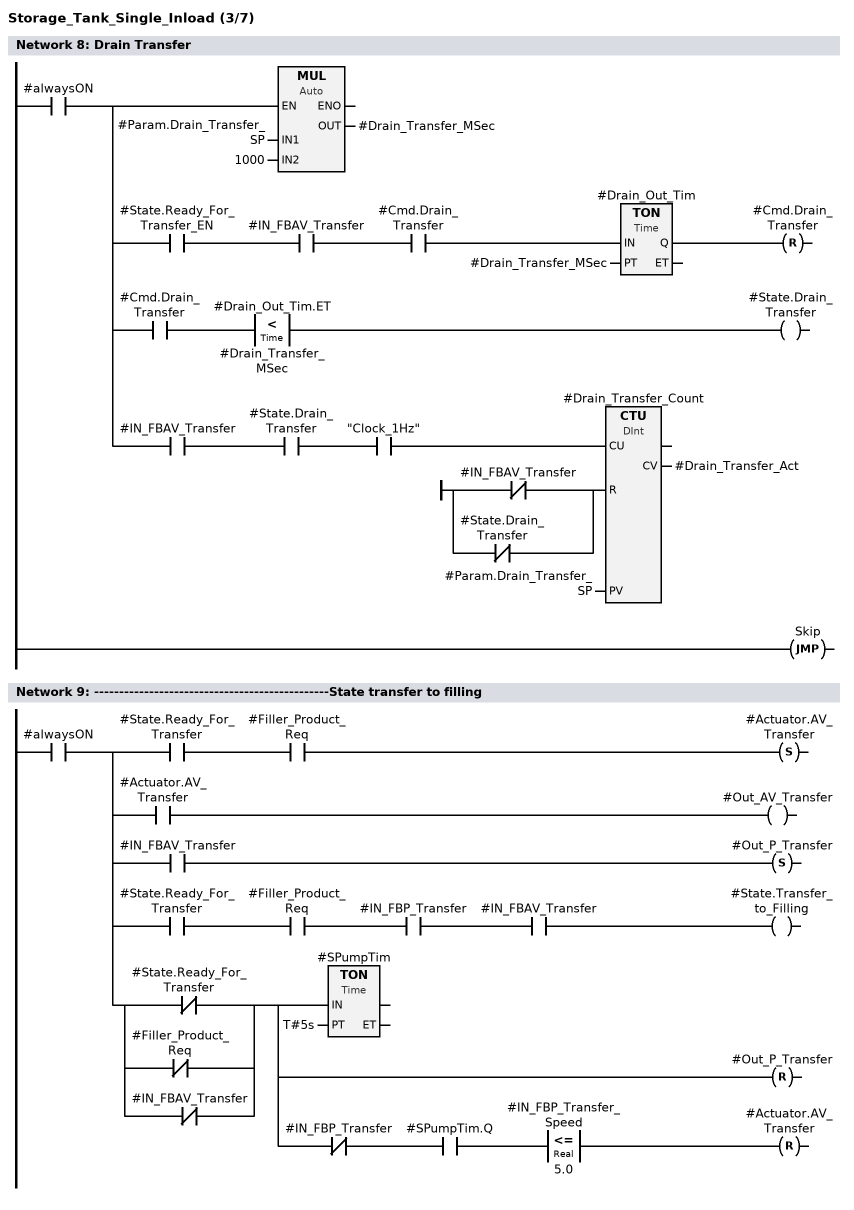
   RUNG wire#powerrail
      Contact( #alwaysON )
      wire#w1
      Mul(in1 := #Param.Drain_Transfer_SP, in2 := 1000, out => #Drain_Transfer_MSec)
   END_RUNG
   RUNG wire#w1
      Contact( #State.Ready_For_Transfer_EN )
      Contact( #IN_FBAV_Transfer )
      Contact( #Cmd.Drain_Transfer )
      { S7_Templates := "time_type := Time" } #Drain_Out_Tim.TON(pt := #Drain_Transfer_MSec, et =>)
      R_Coil( #Cmd.Drain_Transfer )
   END_RUNG
   RUNG wire#w1
      Contact( #Cmd.Drain_Transfer )
      { S7_Templates := "SrcType := Time" } LT_Contact(in1 := #Drain_Out_Tim.ET, in2 := #Drain_Transfer_MSec)
      Coil( #State.Drain_Transfer )
   END_RUNG
   RUNG wire#w1
      Contact( #IN_FBAV_Transfer )
      Contact( #State.Drain_Transfer )
      Contact( "Clock_1Hz" )
      { S7_Templates := "value_type := DInt" } #Drain_Transfer_Count.CTU(r := wire#w2, pv := #Param.Drain_Transfer_SP, cv => #Drain_Transfer_Act)
   END_RUNG
   RUNG wire#powerrail
      I_Contact( #IN_FBAV_Transfer )
   END_RUNG wire#w2
   RUNG wire#powerrail
      I_Contact( #State.Drain_Transfer )
   END_RUNG wire#w2
   RUNG wire#powerrail
      JumpCoil( Skip )
   END_RUNG
   // the same network as SCL:
   IF #alwaysON THEN #Drain_Transfer_MSec := #Param.Drain_Transfer_SP * 1000; END_IF;
   #Drain_Out_Tim(IN := #alwaysON AND #State.Ready_For_Transfer_EN AND #IN_FBAV_Transfer AND #Cmd.Drain_Transfer,   // TON
                  PT := #Drain_Transfer_MSec);
   IF #Drain_Out_Tim.Q THEN #Cmd.Drain_Transfer := FALSE; END_IF;
   #State.Drain_Transfer := #alwaysON AND #Cmd.Drain_Transfer AND (#Drain_Out_Tim.ET < #Drain_Transfer_MSec);
   #Drain_Transfer_Count.CTU(CU := #alwaysON AND #IN_FBAV_Transfer AND #State.Drain_Transfer AND "Clock_1Hz",
                           R := NOT #IN_FBAV_Transfer OR NOT #State.Drain_Transfer,
                           PV := #Param.Drain_Transfer_SP,
                           CV => #Drain_Transfer_Act);
   GOTO Skip;
END_REGION

REGION Network 9: -----------------------------------------------State transfer to filling
   RUNG wire#powerrail
      Contact( #alwaysON )
      wire#w1
      Contact( #State.Ready_For_Transfer )
      Contact( #Filler_Product_Req )
      S_Coil( #Actuator.AV_Transfer )
   END_RUNG
   RUNG wire#w1
      Contact( #Actuator.AV_Transfer )
      Coil( #Out_AV_Transfer )
   END_RUNG
   RUNG wire#w1
      Contact( #IN_FBAV_Transfer )
      S_Coil( #Out_P_Transfer )
   END_RUNG
   RUNG wire#w1
      Contact( #State.Ready_For_Transfer )
      Contact( #Filler_Product_Req )
      Contact( #IN_FBP_Transfer )
      Contact( #IN_FBAV_Transfer )
      Coil( #State.Transfer_to_Filling )
   END_RUNG
   RUNG wire#w1
      I_Contact( #State.Ready_For_Transfer )
      wire#w2
      { S7_Templates := "time_type := Time" } #SPumpTim.TON(pt := T#5s, et =>)
   END_RUNG
   RUNG wire#w1
      I_Contact( #Filler_Product_Req )
   END_RUNG wire#w2
   RUNG wire#w1
      I_Contact( #IN_FBAV_Transfer )
   END_RUNG wire#w2
   RUNG wire#w2
      R_Coil( #Out_P_Transfer )
   END_RUNG
   RUNG wire#w2
      I_Contact( #IN_FBP_Transfer )
      Contact( #SPumpTim.Q )
      { S7_Templates := "SrcType := Real" } LE_Contact(in1 := #IN_FBP_Transfer_Speed, in2 := 5.0)
      R_Coil( #Actuator.AV_Transfer )
   END_RUNG
   // the same network as SCL:
   IF #alwaysON AND #State.Ready_For_Transfer AND #Filler_Product_Req THEN
       #Actuator.AV_Transfer := TRUE;
   END_IF;
   #Out_AV_Transfer := #alwaysON AND #Actuator.AV_Transfer;
   IF #alwaysON AND #IN_FBAV_Transfer THEN #Out_P_Transfer := TRUE; END_IF;
   #State.Transfer_to_Filling := #alwaysON AND #State.Ready_For_Transfer AND #Filler_Product_Req AND #IN_FBP_Transfer AND #IN_FBAV_Transfer;
   #_w1 := #alwaysON AND (NOT #State.Ready_For_Transfer OR NOT #Filler_Product_Req OR NOT #IN_FBAV_Transfer);
   #SPumpTim(IN := #_w1, PT := T#5s);   // TON
   IF #_w1 THEN #Out_P_Transfer := FALSE; END_IF;
   IF #_w1 AND NOT #IN_FBP_Transfer AND #SPumpTim.Q AND (#IN_FBP_Transfer_Speed <= 5.0) THEN
       #Actuator.AV_Transfer := FALSE;
   END_IF;
END_REGION

REGION Network 10: -----------------------------------------------Command CIP
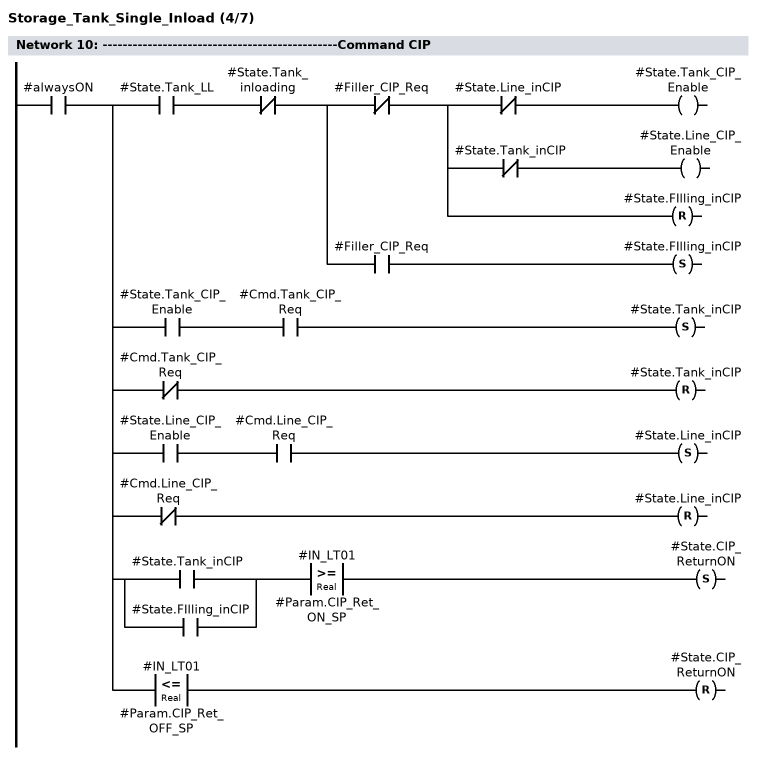
   RUNG wire#powerrail
      Contact( #alwaysON )
      wire#w1
      Contact( #State.Tank_LL )
      I_Contact( #State.Tank_inloading )
      wire#w2
      I_Contact( #Filler_CIP_Req )
      wire#w3
      I_Contact( #State.Line_inCIP )
      Coil( #State.Tank_CIP_Enable )
   END_RUNG
   RUNG wire#w3
      I_Contact( #State.Tank_inCIP )
      Coil( #State.Line_CIP_Enable )
   END_RUNG
   RUNG wire#w3
      R_Coil( #State.FIlling_inCIP )
   END_RUNG
   RUNG wire#w2
      Contact( #Filler_CIP_Req )
      S_Coil( #State.FIlling_inCIP )
   END_RUNG
   RUNG wire#w1
      Contact( #State.Tank_CIP_Enable )
      Contact( #Cmd.Tank_CIP_Req )
      S_Coil( #State.Tank_inCIP )
   END_RUNG
   RUNG wire#w1
      I_Contact( #Cmd.Tank_CIP_Req )
      R_Coil( #State.Tank_inCIP )
   END_RUNG
   RUNG wire#w1
      Contact( #State.Line_CIP_Enable )
      Contact( #Cmd.Line_CIP_Req )
      S_Coil( #State.Line_inCIP )
   END_RUNG
   RUNG wire#w1
      I_Contact( #Cmd.Line_CIP_Req )
      R_Coil( #State.Line_inCIP )
   END_RUNG
   RUNG wire#w1
      Contact( #State.Tank_inCIP )
      wire#w4
      { S7_Templates := "SrcType := Real" } GE_Contact(in1 := #IN_LT01, in2 := #Param.CIP_Ret_ON_SP)
      S_Coil( #State.CIP_ReturnON )
   END_RUNG
   RUNG wire#w1
      Contact( #State.FIlling_inCIP )
   END_RUNG wire#w4
   RUNG wire#w1
      { S7_Templates := "SrcType := Real" } LE_Contact(in1 := #IN_LT01, in2 := #Param.CIP_Ret_OFF_SP)
      R_Coil( #State.CIP_ReturnON )
   END_RUNG
   // the same network as SCL:
   #_w1 := #alwaysON AND #State.Tank_LL AND NOT #State.Tank_inloading;
   #_w2 := #_w1 AND NOT #Filler_CIP_Req;
   #State.Tank_CIP_Enable := #_w2 AND NOT #State.Line_inCIP;
   #State.Line_CIP_Enable := #_w2 AND NOT #State.Tank_inCIP;
   IF #_w2 THEN #State.FIlling_inCIP := FALSE; END_IF;
   IF #_w1 AND #Filler_CIP_Req THEN #State.FIlling_inCIP := TRUE; END_IF;
   IF #alwaysON AND #State.Tank_CIP_Enable AND #Cmd.Tank_CIP_Req THEN #State.Tank_inCIP := TRUE; END_IF;
   IF #alwaysON AND NOT #Cmd.Tank_CIP_Req THEN #State.Tank_inCIP := FALSE; END_IF;
   IF #alwaysON AND #State.Line_CIP_Enable AND #Cmd.Line_CIP_Req THEN #State.Line_inCIP := TRUE; END_IF;
   IF #alwaysON AND NOT #Cmd.Line_CIP_Req THEN #State.Line_inCIP := FALSE; END_IF;
   IF #alwaysON AND (#State.Tank_inCIP OR #State.FIlling_inCIP) AND (#IN_LT01 >= #Param.CIP_Ret_ON_SP) THEN
       #State.CIP_ReturnON := TRUE;
   END_IF;
   IF #alwaysON AND (#IN_LT01 <= #Param.CIP_Ret_OFF_SP) THEN #State.CIP_ReturnON := FALSE; END_IF;
END_REGION

REGION Network 11: Command CIP New
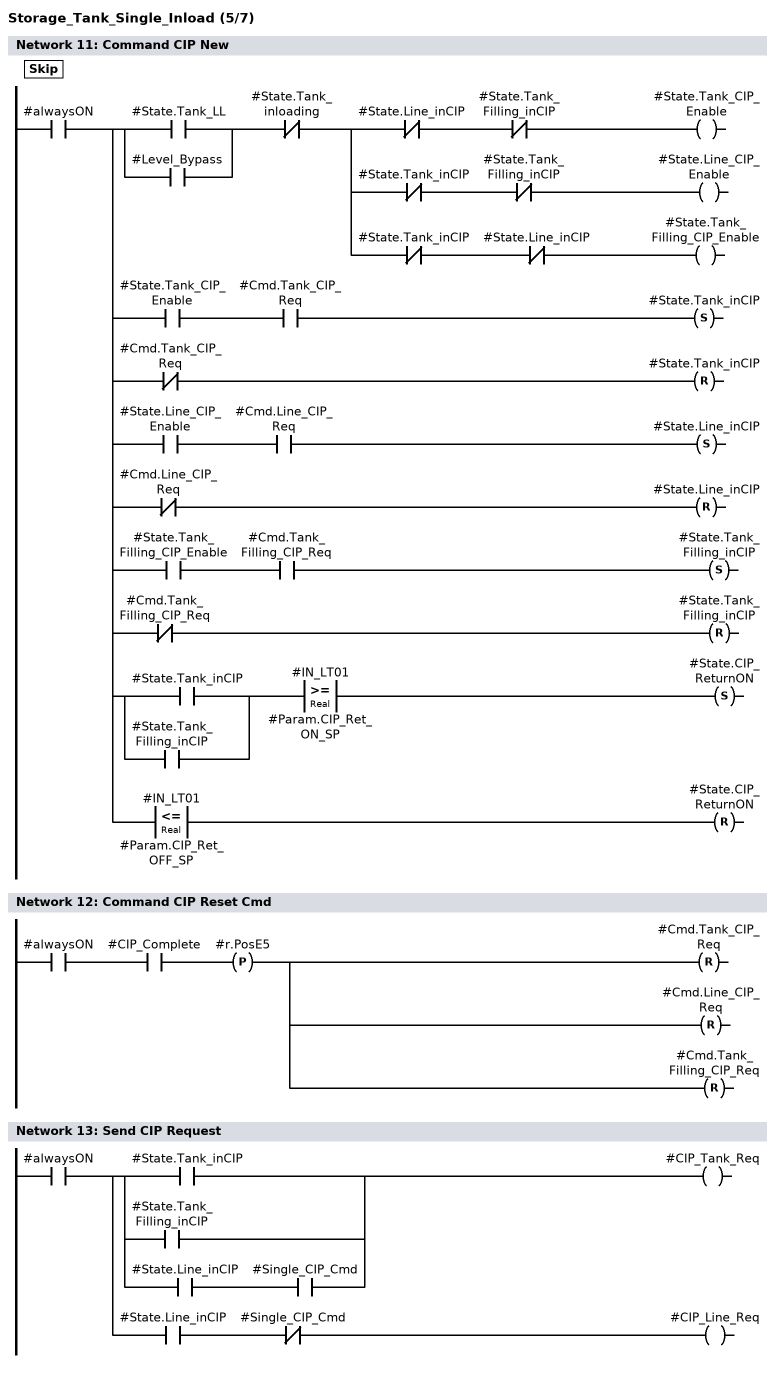
   Label( Skip )
   RUNG wire#powerrail
      Contact( #alwaysON )
      wire#w1
      Contact( #State.Tank_LL )
      wire#w2
      I_Contact( #State.Tank_inloading )
      wire#w3
      I_Contact( #State.Line_inCIP )
      I_Contact( #State.Tank_Filling_inCIP )
      Coil( #State.Tank_CIP_Enable )
   END_RUNG
   RUNG wire#w1
      Contact( #Level_Bypass )
   END_RUNG wire#w2
   RUNG wire#w3
      I_Contact( #State.Tank_inCIP )
      I_Contact( #State.Tank_Filling_inCIP )
      Coil( #State.Line_CIP_Enable )
   END_RUNG
   RUNG wire#w3
      I_Contact( #State.Tank_inCIP )
      I_Contact( #State.Line_inCIP )
      Coil( #State.Tank_Filling_CIP_Enable )
   END_RUNG
   RUNG wire#w1
      Contact( #State.Tank_CIP_Enable )
      Contact( #Cmd.Tank_CIP_Req )
      S_Coil( #State.Tank_inCIP )
   END_RUNG
   RUNG wire#w1
      I_Contact( #Cmd.Tank_CIP_Req )
      R_Coil( #State.Tank_inCIP )
   END_RUNG
   RUNG wire#w1
      Contact( #State.Line_CIP_Enable )
      Contact( #Cmd.Line_CIP_Req )
      S_Coil( #State.Line_inCIP )
   END_RUNG
   RUNG wire#w1
      I_Contact( #Cmd.Line_CIP_Req )
      R_Coil( #State.Line_inCIP )
   END_RUNG
   RUNG wire#w1
      Contact( #State.Tank_Filling_CIP_Enable )
      Contact( #Cmd.Tank_Filling_CIP_Req )
      S_Coil( #State.Tank_Filling_inCIP )
   END_RUNG
   RUNG wire#w1
      I_Contact( #Cmd.Tank_Filling_CIP_Req )
      R_Coil( #State.Tank_Filling_inCIP )
   END_RUNG
   RUNG wire#w1
      Contact( #State.Tank_inCIP )
      wire#w4
      { S7_Templates := "SrcType := Real" } GE_Contact(in1 := #IN_LT01, in2 := #Param.CIP_Ret_ON_SP)
      S_Coil( #State.CIP_ReturnON )
   END_RUNG
   RUNG wire#w1
      Contact( #State.Tank_Filling_inCIP )
   END_RUNG wire#w4
   RUNG wire#w1
      { S7_Templates := "SrcType := Real" } LE_Contact(in1 := #IN_LT01, in2 := #Param.CIP_Ret_OFF_SP)
      R_Coil( #State.CIP_ReturnON )
   END_RUNG
   // the same network as SCL:
   Skip:
   #_w1 := #alwaysON AND (#State.Tank_LL OR #Level_Bypass) AND NOT #State.Tank_inloading;
   #State.Tank_CIP_Enable := #_w1 AND NOT #State.Line_inCIP AND NOT #State.Tank_Filling_inCIP;
   #State.Line_CIP_Enable := #_w1 AND NOT #State.Tank_inCIP AND NOT #State.Tank_Filling_inCIP;
   #State.Tank_Filling_CIP_Enable := #_w1 AND NOT #State.Tank_inCIP AND NOT #State.Line_inCIP;
   IF #alwaysON AND #State.Tank_CIP_Enable AND #Cmd.Tank_CIP_Req THEN #State.Tank_inCIP := TRUE; END_IF;
   IF #alwaysON AND NOT #Cmd.Tank_CIP_Req THEN #State.Tank_inCIP := FALSE; END_IF;
   IF #alwaysON AND #State.Line_CIP_Enable AND #Cmd.Line_CIP_Req THEN #State.Line_inCIP := TRUE; END_IF;
   IF #alwaysON AND NOT #Cmd.Line_CIP_Req THEN #State.Line_inCIP := FALSE; END_IF;
   IF #alwaysON AND #State.Tank_Filling_CIP_Enable AND #Cmd.Tank_Filling_CIP_Req THEN
       #State.Tank_Filling_inCIP := TRUE;
   END_IF;
   IF #alwaysON AND NOT #Cmd.Tank_Filling_CIP_Req THEN #State.Tank_Filling_inCIP := FALSE; END_IF;
   IF #alwaysON AND (#State.Tank_inCIP OR #State.Tank_Filling_inCIP) AND (#IN_LT01 >= #Param.CIP_Ret_ON_SP) THEN
       #State.CIP_ReturnON := TRUE;
   END_IF;
   IF #alwaysON AND (#IN_LT01 <= #Param.CIP_Ret_OFF_SP) THEN #State.CIP_ReturnON := FALSE; END_IF;
END_REGION

REGION Network 12: Command CIP Reset Cmd
   RUNG wire#powerrail
      Contact( #alwaysON )
      Contact( #CIP_Complete )
      P_Trig( #r.PosE5 )
      wire#w1
      R_Coil( #Cmd.Tank_CIP_Req )
   END_RUNG
   RUNG wire#w1
      R_Coil( #Cmd.Line_CIP_Req )
   END_RUNG
   RUNG wire#w1
      R_Coil( #Cmd.Tank_Filling_CIP_Req )
   END_RUNG
   // the same network as SCL:
   #_w1 := #alwaysON AND #CIP_Complete;
   #_w2 := #_w1 AND NOT #r.PosE5;   // rising edge
   #r.PosE5 := #_w1;
   IF #_w2 THEN
       #Cmd.Tank_CIP_Req := FALSE;
       #Cmd.Line_CIP_Req := FALSE;
       #Cmd.Tank_Filling_CIP_Req := FALSE;
   END_IF;
END_REGION

REGION Network 13: Send CIP Request
   RUNG wire#powerrail
      Contact( #alwaysON )
      wire#w1
      Contact( #State.Tank_inCIP )
      wire#w2
      Coil( #CIP_Tank_Req )
   END_RUNG
   RUNG wire#w1
      Contact( #State.Tank_Filling_inCIP )
   END_RUNG wire#w2
   RUNG wire#w1
      Contact( #State.Line_inCIP )
      Contact( #Single_CIP_Cmd )
   END_RUNG wire#w2
   RUNG wire#w1
      Contact( #State.Line_inCIP )
      I_Contact( #Single_CIP_Cmd )
      Coil( #CIP_Line_Req )
   END_RUNG
   // the same network as SCL:
   #CIP_Tank_Req := #alwaysON AND (#State.Tank_inCIP OR #State.Tank_Filling_inCIP OR (#State.Line_inCIP AND #Single_CIP_Cmd));
   #CIP_Line_Req := #alwaysON AND #State.Line_inCIP AND NOT #Single_CIP_Cmd;
END_REGION

REGION Network 14: Send CIP Line OK
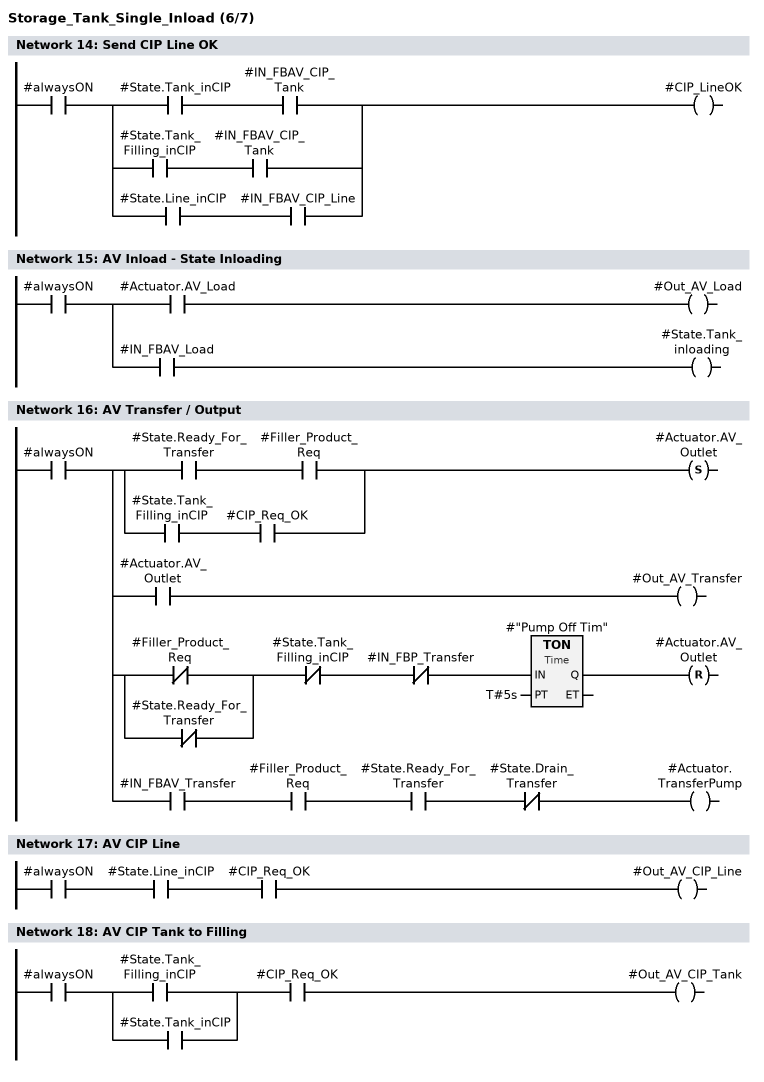
   RUNG wire#powerrail
      Contact( #alwaysON )
      wire#w1
      Contact( #State.Tank_inCIP )
      Contact( #IN_FBAV_CIP_Tank )
      wire#w2
      Coil( #CIP_LineOK )
   END_RUNG
   RUNG wire#w1
      Contact( #State.Tank_Filling_inCIP )
      Contact( #IN_FBAV_CIP_Tank )
   END_RUNG wire#w2
   RUNG wire#w1
      Contact( #State.Line_inCIP )
      Contact( #IN_FBAV_CIP_Line )
   END_RUNG wire#w2
   // the same network as SCL:
   #CIP_LineOK := #alwaysON AND ((#State.Tank_inCIP AND #IN_FBAV_CIP_Tank) OR (#State.Tank_Filling_inCIP AND #IN_FBAV_CIP_Tank) OR (#State.Line_inCIP AND #IN_FBAV_CIP_Line));
END_REGION

REGION Network 15: AV Inload - State Inloading
   RUNG wire#powerrail
      Contact( #alwaysON )
      wire#w1
      Contact( #Actuator.AV_Load )
      Coil( #Out_AV_Load )
   END_RUNG
   RUNG wire#w1
      Contact( #IN_FBAV_Load )
      Coil( #State.Tank_inloading )
   END_RUNG
   // the same network as SCL:
   #Out_AV_Load := #alwaysON AND #Actuator.AV_Load;
   #State.Tank_inloading := #alwaysON AND #IN_FBAV_Load;
END_REGION

REGION Network 16: AV Transfer / Output
   RUNG wire#powerrail
      Contact( #alwaysON )
      wire#w1
      Contact( #State.Ready_For_Transfer )
      Contact( #Filler_Product_Req )
      wire#w2
      S_Coil( #Actuator.AV_Outlet )
   END_RUNG
   RUNG wire#w1
      Contact( #State.Tank_Filling_inCIP )
      Contact( #CIP_Req_OK )
   END_RUNG wire#w2
   RUNG wire#w1
      Contact( #Actuator.AV_Outlet )
      Coil( #Out_AV_Transfer )
   END_RUNG
   RUNG wire#w1
      I_Contact( #Filler_Product_Req )
      wire#w3
      I_Contact( #State.Tank_Filling_inCIP )
      I_Contact( #IN_FBP_Transfer )
      { S7_Templates := "time_type := Time" } #"Pump Off Tim".TON(pt := T#5s, et =>)
      R_Coil( #Actuator.AV_Outlet )
   END_RUNG
   RUNG wire#w1
      I_Contact( #State.Ready_For_Transfer )
   END_RUNG wire#w3
   RUNG wire#w1
      Contact( #IN_FBAV_Transfer )
      Contact( #Filler_Product_Req )
      Contact( #State.Ready_For_Transfer )
      I_Contact( #State.Drain_Transfer )
      Coil( #Actuator.TransferPump )
   END_RUNG
   // the same network as SCL:
   IF #alwaysON AND ((#State.Ready_For_Transfer AND #Filler_Product_Req) OR (#State.Tank_Filling_inCIP AND #CIP_Req_OK)) THEN
       #Actuator.AV_Outlet := TRUE;
   END_IF;
   #Out_AV_Transfer := #alwaysON AND #Actuator.AV_Outlet;
   #"Pump Off Tim"(IN := #alwaysON AND (NOT #Filler_Product_Req OR NOT #State.Ready_For_Transfer) AND NOT #State.Tank_Filling_inCIP AND NOT #IN_FBP_Transfer,   // TON
                   PT := T#5s);
   IF #"Pump Off Tim".Q THEN #Actuator.AV_Outlet := FALSE; END_IF;
   #Actuator.TransferPump := #alwaysON AND #IN_FBAV_Transfer AND #Filler_Product_Req AND #State.Ready_For_Transfer AND NOT #State.Drain_Transfer;
END_REGION

REGION Network 17: AV CIP Line
   RUNG wire#powerrail
      Contact( #alwaysON )
      Contact( #State.Line_inCIP )
      Contact( #CIP_Req_OK )
      Coil( #Out_AV_CIP_Line )
   END_RUNG
   // the same network as SCL:
   #Out_AV_CIP_Line := #alwaysON AND #State.Line_inCIP AND #CIP_Req_OK;
END_REGION

REGION Network 18: AV CIP Tank to Filling
   RUNG wire#powerrail
      Contact( #alwaysON )
      wire#w1
      Contact( #State.Tank_Filling_inCIP )
      wire#w2
      Contact( #CIP_Req_OK )
      Coil( #Out_AV_CIP_Tank )
   END_RUNG
   RUNG wire#w1
      Contact( #State.Tank_inCIP )
   END_RUNG wire#w2
   // the same network as SCL:
   #Out_AV_CIP_Tank := #alwaysON AND (#State.Tank_Filling_inCIP OR #State.Tank_inCIP) AND #CIP_Req_OK;
END_REGION

REGION Network 19: Pump Transfer
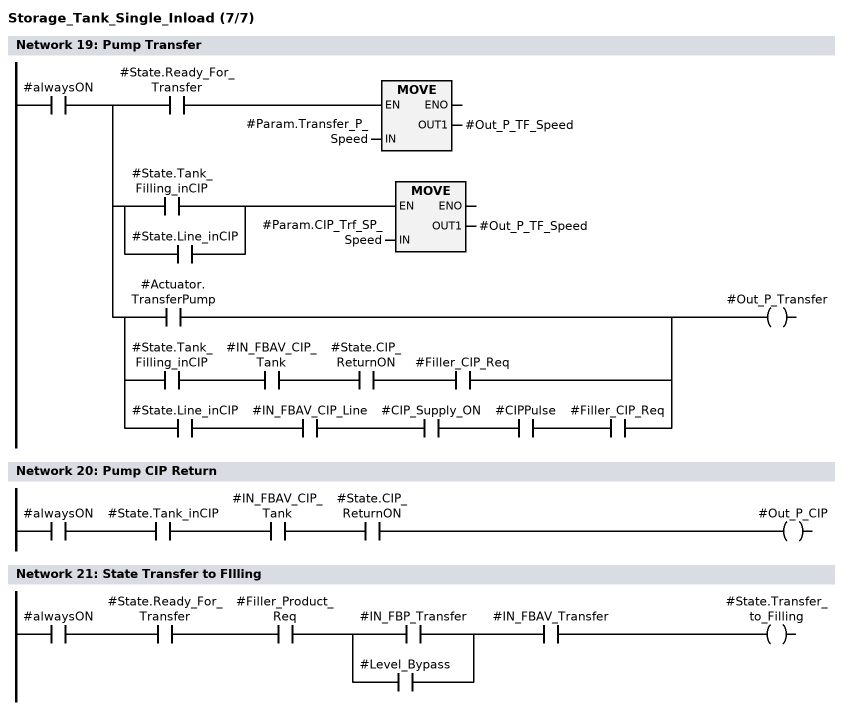
   RUNG wire#powerrail
      Contact( #alwaysON )
      wire#w1
      Contact( #State.Ready_For_Transfer )
      Move(in := #Param.Transfer_P_Speed, out1 => #Out_P_TF_Speed)
   END_RUNG
   RUNG wire#w1
      Contact( #State.Tank_Filling_inCIP )
      wire#w2
      Move(in := #Param.CIP_Trf_SP_Speed, out1 => #Out_P_TF_Speed)
   END_RUNG
   RUNG wire#w1
      Contact( #State.Line_inCIP )
   END_RUNG wire#w2
   RUNG wire#w1
      Contact( #Actuator.TransferPump )
      wire#w3
      Coil( #Out_P_Transfer )
   END_RUNG
   RUNG wire#w1
      Contact( #State.Tank_Filling_inCIP )
      Contact( #IN_FBAV_CIP_Tank )
      Contact( #State.CIP_ReturnON )
      Contact( #Filler_CIP_Req )
   END_RUNG wire#w3
   RUNG wire#w1
      Contact( #State.Line_inCIP )
      Contact( #IN_FBAV_CIP_Line )
      Contact( #CIP_Supply_ON )
      Contact( #CIPPulse )
      Contact( #Filler_CIP_Req )
   END_RUNG wire#w3
   // the same network as SCL:
   IF #alwaysON AND #State.Ready_For_Transfer THEN #Out_P_TF_Speed := #Param.Transfer_P_Speed; END_IF;
   IF #alwaysON AND (#State.Tank_Filling_inCIP OR #State.Line_inCIP) THEN
       #Out_P_TF_Speed := #Param.CIP_Trf_SP_Speed;
   END_IF;
   #Out_P_Transfer := #alwaysON AND (#Actuator.TransferPump OR (#State.Tank_Filling_inCIP AND #IN_FBAV_CIP_Tank AND #State.CIP_ReturnON AND #Filler_CIP_Req) OR (#State.Line_inCIP AND #IN_FBAV_CIP_Line AND #CIP_Supply_ON AND #CIPPulse AND #Filler_CIP_Req));
END_REGION

REGION Network 20: Pump CIP Return
   RUNG wire#powerrail
      Contact( #alwaysON )
      Contact( #State.Tank_inCIP )
      Contact( #IN_FBAV_CIP_Tank )
      Contact( #State.CIP_ReturnON )
      Coil( #Out_P_CIP )
   END_RUNG
   // the same network as SCL:
   #Out_P_CIP := #alwaysON AND #State.Tank_inCIP AND #IN_FBAV_CIP_Tank AND #State.CIP_ReturnON;
END_REGION

REGION Network 21: State Transfer to FIlling
   RUNG wire#powerrail
      Contact( #alwaysON )
      Contact( #State.Ready_For_Transfer )
      Contact( #Filler_Product_Req )
      wire#w1
      Contact( #IN_FBP_Transfer )
      wire#w2
      Contact( #IN_FBAV_Transfer )
      Coil( #State.Transfer_to_Filling )
   END_RUNG
   RUNG wire#w1
      Contact( #Level_Bypass )
   END_RUNG wire#w2
   // the same network as SCL:
   #State.Transfer_to_Filling := #alwaysON AND #State.Ready_For_Transfer AND #Filler_Product_Req AND (#IN_FBP_Transfer OR #Level_Bypass) AND #IN_FBAV_Transfer;
END_REGION
END_FUNCTION_BLOCK

FUNCTION_BLOCK "Storage_Tank_Multi_Inload"   // FB23, LAD
{ S7_Optimized_Access := 'FALSE' }
VERSION : 0.1
// stored: AutoNumber false, IsIECCheckEnabled false, SetENOAutomatically false, UDAEnableTagReadback false
   VAR_INPUT
      Level_Bypass : Bool;
      Single_CIP_Cmd : Bool;
      IN_FBAV_Load : Bool;
      IN_FBAV_Transfer : Bool;
      IN_FBP_Transfer : Bool;
      IN_FBP_Transfer_Speed : Real;
      IN_FBP_CIP : Bool;
      IN_FBAV_CIP_Sup : Bool;
      IN_FBAV_CIP_Tank : Bool;
      IN_FBAV_CIP_Line : Bool;
      IN_LT01 : Real;
      IN_FS : Bool;
      CIP_Req_OK : Bool;
      CIP_ON_Progress : Bool;
      CIP_Supply_ON : Bool;
      CIP_Complete : Bool;
      CIPPulse : Bool;
      Filler_Product_Req : Bool;
      Filler_CIP_Req : Bool;
      Loading_Busy_1 : Bool;
      Loading_Busy_2 : Bool;
      Loading_Busy_3 : Bool;
      Transfer_Busy : Bool;
      CIP_En : Bool;
   END_VAR
   VAR_OUTPUT
      Out_AV_Load : Bool;
      Out_AV_Transfer : Bool;
      Out_P_Transfer : Bool;
      Out_P_TF_Speed : Real;
      Out_P_CIP : Bool;
      Out_AV_CIP_Line : Bool;
      Out_AV_CIP_Tank : Bool;
      Out_AV_CIP_Filling : Bool;
      CIP_Tank_Req : Bool;
      CIP_Line_Req : Bool;
      CIP_LineOK : Bool;
   END_VAR
   VAR DB_SPECIFIC
      Cmd : Struct
         Inload_Select_Tank_1 : Bool;
         Inload_Select_Tank_2 : Bool;
         Inload_Select_Tank_3 : Bool;
         Inload : Bool;   // Start Loading
         Tank_CIP_Req : Bool;
         Line_CIP_Req : Bool;
         Tank_Filling_CIP_Req : Bool;
         CIP_Filling_En : Bool;
         CIP_Line_Req_OK : Bool;
         CIP_Supply_ON : Bool;
         CIP_ON_Progress : Bool;
         Flushing : Bool;   // Water Flushing
         RaadyForTF : Bool;   // Tank Ready for Blending
         Flush_Select : Byte;
         Drain_In : Bool;
         Drain_Transfer : Bool;
      END_STRUCT;
      Param : Struct
         SP_Level_LL : Real := 10.0;
         SP_Level_ML : Real := 80.0;
         SP_Level_HL : Real := 100.0;
         SupplyPump_SP_Speed : Real := 80.0;
         L_Hi_Lim : Real := 100.0;
         L_Lo_Lim : Real := 0.0;
         L_Hys : Real := 2.0;
         FlushingTime : DInt := 10000;
         CIP_Trf_SP_Speed : Real := 80.0;
         CIP_Ret_ON_SP : Real := 10.0;
         CIP_Ret_OFF_SP : Real;
         Transfer_P_Speed : Real := 60.0;
         Drain_Inload_SP : DInt := 10;
         Drain_Transfer_SP : DInt := 10;
         SP_Agi_On : Real := 20.0;
      END_STRUCT;
      State : Struct   // Tank in loading state
         Tank_inloading : Bool;
         Tank_inCIP : Bool;
         Tank_Filling_inCIP : Bool;
         Line_inCIP : Bool;
         FIlling_inCIP : Bool;
         Flushing : Bool;
         Tank_LL : Bool;
         Tank_ML : Bool;
         Tank_HL : Bool;
         Inload_Enable : Bool;
         Tank_CIP_Enable : Bool;
         Line_CIP_Enable : Bool;
         Tank_Filling_CIP_Enable : Bool;
         Flushing_Enable : Bool;
         Flush_selected : Byte;
         CIP_Request_OK : Bool;
         CIP_ReturnON : Bool;
         Ready_For_Transfer_EN : Bool;   // Tank Ready for Transfer to Blending
         Ready_For_Transfer : Bool;   // Tank Ready for Transfer to Blending
         HWT_Status : Int;
         Transfer_to_Filling : Bool;
         "Line_AV4&AV5" : Bool;
         "Line_AV1&AV2" : Bool;
         "Line_AV7&AV8" : Bool;
         "Line_AV10&AV11" : Bool;
         "Line_AV5&AV6" : Bool;
         CIP_Line1_ON : Bool;
         CIP_Line2_ON : Bool;
         CIP_Line3_ON : Bool;
         CIP_Line4_ON : Bool;
         Drain_Inload : Bool;
         Drain_Transfer : Bool;
         Agi_ON : Bool;
         "CIP Req" : Bool;
      END_STRUCT;
      alwaysON : Bool;
      L_Hys_Abs : Real;
      Hys_Level_HL : Real;
      Hys_Level_ML : Real;
      Hys_Level_LL : Real;
      Drain_Inload_MSec : DInt;
      Drain_Inload_Count : IEC_DCOUNTER;
      Drain_Inload_Act { S7_SetPoint := 'True'} : DInt;
      Drain_Transfer_MSec : DInt;
      Drain_Transfer_Count : IEC_DCOUNTER;
      Drain_Transfer_Act : DInt;
      r : Struct
         PosE1 : Bool;
         PosE2 : Bool;
         PosE3 : Bool;
         PosE4 : Bool;
         PosE5 : Bool;
         PosE6 : Bool;
         PosE7 : Bool;
         PosE8 : Bool;
         PosE9 : Bool;
         PosE10 : Bool;
         PosE11 : Bool;
         PosE12 : Bool;
         PosE13 : Bool;
         PosE14 : Bool;
         PosE15 : Bool;
         PosE16 : Bool;
         PosE17 : Bool;
         PosE18 : Bool;
         PosE19 : Bool;
         PosE20 : Bool;
         PosE21 : Bool;
         PosE22 : Bool;
         PosE23 : Bool;
         PosE24 : Bool;
         PosE25 : Bool;
         PosE26 : Bool;
         PosE27 : Bool;
         PosE28 : Bool;
         PosE29 : Bool;
         PosE30 : Bool;
         PosE31 : Bool;
         PosE32 : Bool;
      END_STRUCT;
      Actuator : Struct
         AV_Outlet : Bool;
         AV_Load : Bool;
         AV_Transfer : Bool;
         CIP_Line_Pump : Bool;
         CIP_Tank_Pump : Bool;
         TransferPump : Bool;
         FlushPump : Bool;
         CV_Steam : Bool;
         Pump : Bool;
      END_STRUCT;
      SPumpTim { S7_SetPoint := 'True'} : TON_TIME;
      SAV_CIPLine { S7_SetPoint := 'True'} : TON_TIME;
      SAV_CIPTANK { S7_SetPoint := 'True'} : TON_TIME;
      SAV_CIPFILLING { S7_SetPoint := 'True'} : TON_TIME;
      AVinloadTim { S7_SetPoint := 'True'} : TON_TIME;
      AVOutletTim { S7_SetPoint := 'True'} : TON_TIME;
      Drain_In_Tim { S7_SetPoint := 'True'} : TON_TIME;
      Drain_Out_Tim { S7_SetPoint := 'True'} : TON_TIME;
      "Pump Off Tim" { S7_SetPoint := 'True'} : TON_TIME;
      "Loading_Busy Tim_1" { S7_SetPoint := 'True'} : TON_TIME;
      "Loading_Busy Tim_2" { S7_SetPoint := 'True'} : TON_TIME;
      "Loading_Busy Tim_3" { S7_SetPoint := 'True'} : TON_TIME;
      Hys_Level_Agi { S7_SetPoint := 'True'} : Real;
   END_VAR
   VAR_TEMP   // added for the SCL form of the ladder/FBD networks
      _w1 : Bool;
      _w2 : Bool;
      _w3 : Bool;
      _w4 : Bool;
      _w5 : Bool;
   END_VAR
BEGIN

REGION Network 1: Always ON
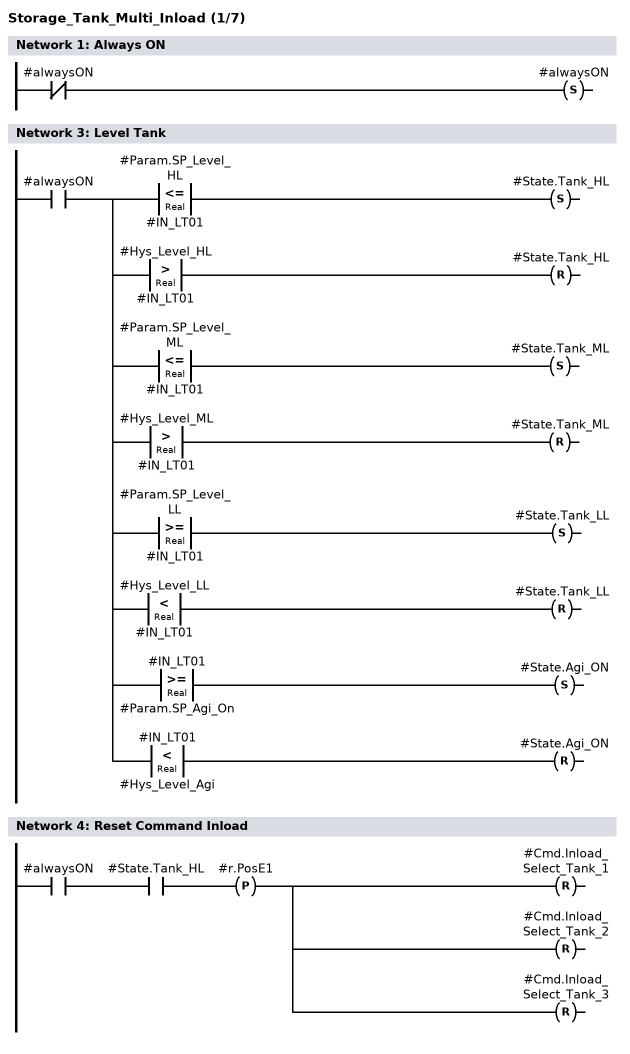
   RUNG wire#powerrail
      I_Contact( #alwaysON )
      S_Coil( #alwaysON )
   END_RUNG
   // the same network as SCL:
   IF NOT #alwaysON THEN #alwaysON := TRUE; END_IF;
END_REGION

NETWORK
TITLE = Hys Calculation
//Level Hys Absolute
      L     #Param.L_Hi_Lim;
      L     #Param.L_Lo_Lim;
      -R;
      L     100.0;
      /R;
      L     #Param.L_Hys;
      *R;
      T     #L_Hys_Abs;
//Tank High Level
      L     #Param.SP_Level_HL;
      L     #L_Hys_Abs;
      -R;
      T     #Hys_Level_HL;
//Tank Mid Level
      L     #Param.SP_Level_ML;
      L     #L_Hys_Abs;
      -R;
      T     #Hys_Level_ML;
//Tank Low Level
      L     #Param.SP_Level_LL;
      L     #L_Hys_Abs;
      +R;
      T     #Hys_Level_LL;
//Level Agi On
      L     #Param.SP_Agi_On;
      L     #L_Hys_Abs;
      -R;
      T     #Hys_Level_Agi;




REGION Network 3: Level Tank
   RUNG wire#powerrail
      Contact( #alwaysON )
      wire#w1
      { S7_Templates := "SrcType := Real" } LE_Contact(in1 := #Param.SP_Level_HL, in2 := #IN_LT01)
      S_Coil( #State.Tank_HL )
   END_RUNG
   RUNG wire#w1
      { S7_Templates := "SrcType := Real" } GT_Contact(in1 := #Hys_Level_HL, in2 := #IN_LT01)
      R_Coil( #State.Tank_HL )
   END_RUNG
   RUNG wire#w1
      { S7_Templates := "SrcType := Real" } LE_Contact(in1 := #Param.SP_Level_ML, in2 := #IN_LT01)
      S_Coil( #State.Tank_ML )
   END_RUNG
   RUNG wire#w1
      { S7_Templates := "SrcType := Real" } GT_Contact(in1 := #Hys_Level_ML, in2 := #IN_LT01)
      R_Coil( #State.Tank_ML )
   END_RUNG
   RUNG wire#w1
      { S7_Templates := "SrcType := Real" } GE_Contact(in1 := #Param.SP_Level_LL, in2 := #IN_LT01)
      S_Coil( #State.Tank_LL )
   END_RUNG
   RUNG wire#w1
      { S7_Templates := "SrcType := Real" } LT_Contact(in1 := #Hys_Level_LL, in2 := #IN_LT01)
      R_Coil( #State.Tank_LL )
   END_RUNG
   RUNG wire#w1
      { S7_Templates := "SrcType := Real" } GE_Contact(in1 := #IN_LT01, in2 := #Param.SP_Agi_On)
      S_Coil( #State.Agi_ON )
   END_RUNG
   RUNG wire#w1
      { S7_Templates := "SrcType := Real" } LT_Contact(in1 := #IN_LT01, in2 := #Hys_Level_Agi)
      R_Coil( #State.Agi_ON )
   END_RUNG
   // the same network as SCL:
   IF #alwaysON AND (#Param.SP_Level_HL <= #IN_LT01) THEN #State.Tank_HL := TRUE; END_IF;
   IF #alwaysON AND (#Hys_Level_HL > #IN_LT01) THEN #State.Tank_HL := FALSE; END_IF;
   IF #alwaysON AND (#Param.SP_Level_ML <= #IN_LT01) THEN #State.Tank_ML := TRUE; END_IF;
   IF #alwaysON AND (#Hys_Level_ML > #IN_LT01) THEN #State.Tank_ML := FALSE; END_IF;
   IF #alwaysON AND (#Param.SP_Level_LL >= #IN_LT01) THEN #State.Tank_LL := TRUE; END_IF;
   IF #alwaysON AND (#Hys_Level_LL < #IN_LT01) THEN #State.Tank_LL := FALSE; END_IF;
   IF #alwaysON AND (#IN_LT01 >= #Param.SP_Agi_On) THEN #State.Agi_ON := TRUE; END_IF;
   IF #alwaysON AND (#IN_LT01 < #Hys_Level_Agi) THEN #State.Agi_ON := FALSE; END_IF;
END_REGION

REGION Network 4: Reset Command Inload
   RUNG wire#powerrail
      Contact( #alwaysON )
      Contact( #State.Tank_HL )
      P_Trig( #r.PosE1 )
      wire#w1
      R_Coil( #Cmd.Inload_Select_Tank_1 )
   END_RUNG
   RUNG wire#w1
      R_Coil( #Cmd.Inload_Select_Tank_2 )
   END_RUNG
   RUNG wire#w1
      R_Coil( #Cmd.Inload_Select_Tank_3 )
   END_RUNG
   // the same network as SCL:
   #_w1 := #alwaysON AND #State.Tank_HL;
   #_w2 := #_w1 AND NOT #r.PosE1;   // rising edge
   #r.PosE1 := #_w1;
   IF #_w2 THEN
       #Cmd.Inload_Select_Tank_1 := FALSE;
       #Cmd.Inload_Select_Tank_2 := FALSE;
       #Cmd.Inload_Select_Tank_3 := FALSE;
   END_IF;
END_REGION

REGION Network 5: Command Inload
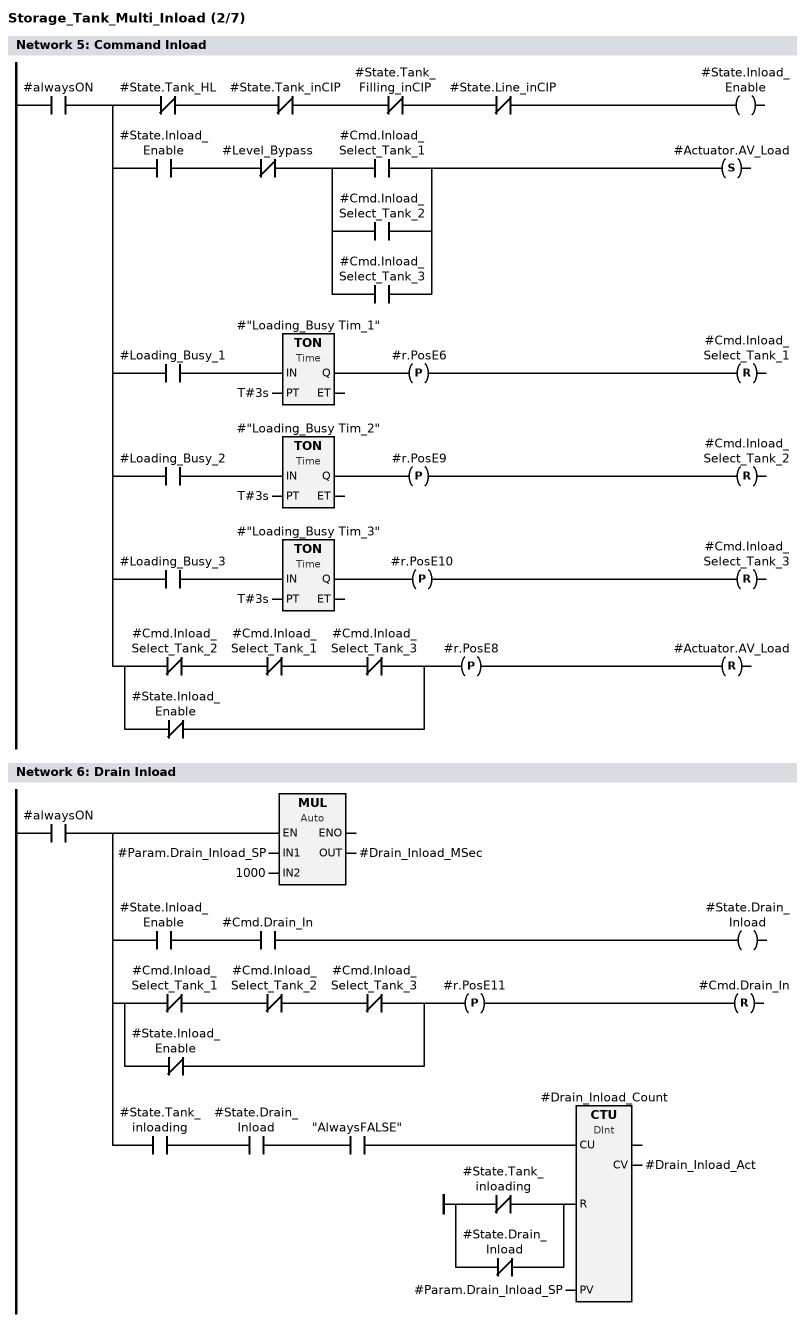
   RUNG wire#powerrail
      Contact( #alwaysON )
      wire#w1
      I_Contact( #State.Tank_HL )
      I_Contact( #State.Tank_inCIP )
      I_Contact( #State.Tank_Filling_inCIP )
      I_Contact( #State.Line_inCIP )
      Coil( #State.Inload_Enable )
   END_RUNG
   RUNG wire#w1
      Contact( #State.Inload_Enable )
      I_Contact( #Level_Bypass )
      wire#w2
      Contact( #Cmd.Inload_Select_Tank_1 )
      wire#w3
      S_Coil( #Actuator.AV_Load )
   END_RUNG
   RUNG wire#w2
      Contact( #Cmd.Inload_Select_Tank_2 )
   END_RUNG wire#w3
   RUNG wire#w2
      Contact( #Cmd.Inload_Select_Tank_3 )
   END_RUNG wire#w3
   RUNG wire#w1
      Contact( #Loading_Busy_1 )
      { S7_Templates := "time_type := Time" } #"Loading_Busy Tim_1".TON(pt := T#3s, et =>)
      P_Trig( #r.PosE6 )
      R_Coil( #Cmd.Inload_Select_Tank_1 )
   END_RUNG
   RUNG wire#w1
      Contact( #Loading_Busy_2 )
      { S7_Templates := "time_type := Time" } #"Loading_Busy Tim_2".TON(pt := T#3s, et =>)
      P_Trig( #r.PosE9 )
      R_Coil( #Cmd.Inload_Select_Tank_2 )
   END_RUNG
   RUNG wire#w1
      Contact( #Loading_Busy_3 )
      { S7_Templates := "time_type := Time" } #"Loading_Busy Tim_3".TON(pt := T#3s, et =>)
      P_Trig( #r.PosE10 )
      R_Coil( #Cmd.Inload_Select_Tank_3 )
   END_RUNG
   RUNG wire#w1
      I_Contact( #Cmd.Inload_Select_Tank_2 )
      I_Contact( #Cmd.Inload_Select_Tank_1 )
      I_Contact( #Cmd.Inload_Select_Tank_3 )
      wire#w4
      P_Trig( #r.PosE8 )
      R_Coil( #Actuator.AV_Load )
   END_RUNG
   RUNG wire#w1
      I_Contact( #State.Inload_Enable )
   END_RUNG wire#w4
   // the same network as SCL:
   #State.Inload_Enable := #alwaysON AND NOT #State.Tank_HL AND NOT #State.Tank_inCIP AND NOT #State.Tank_Filling_inCIP AND NOT #State.Line_inCIP;
   IF #alwaysON AND #State.Inload_Enable AND NOT #Level_Bypass AND (#Cmd.Inload_Select_Tank_1 OR #Cmd.Inload_Select_Tank_2 OR #Cmd.Inload_Select_Tank_3) THEN
       #Actuator.AV_Load := TRUE;
   END_IF;
   #"Loading_Busy Tim_1"(IN := #alwaysON AND #Loading_Busy_1, PT := T#3s);   // TON
   #_w1 := #"Loading_Busy Tim_1".Q AND NOT #r.PosE6;   // rising edge
   #r.PosE6 := #"Loading_Busy Tim_1".Q;
   IF #_w1 THEN #Cmd.Inload_Select_Tank_1 := FALSE; END_IF;
   #"Loading_Busy Tim_2"(IN := #alwaysON AND #Loading_Busy_2, PT := T#3s);   // TON
   #_w2 := #"Loading_Busy Tim_2".Q AND NOT #r.PosE9;   // rising edge
   #r.PosE9 := #"Loading_Busy Tim_2".Q;
   IF #_w2 THEN #Cmd.Inload_Select_Tank_2 := FALSE; END_IF;
   #"Loading_Busy Tim_3"(IN := #alwaysON AND #Loading_Busy_3, PT := T#3s);   // TON
   #_w3 := #"Loading_Busy Tim_3".Q AND NOT #r.PosE10;   // rising edge
   #r.PosE10 := #"Loading_Busy Tim_3".Q;
   IF #_w3 THEN #Cmd.Inload_Select_Tank_3 := FALSE; END_IF;
   #_w4 := #alwaysON AND ((NOT #Cmd.Inload_Select_Tank_2 AND NOT #Cmd.Inload_Select_Tank_1 AND NOT #Cmd.Inload_Select_Tank_3) OR NOT #State.Inload_Enable);
   #_w5 := #_w4 AND NOT #r.PosE8;   // rising edge
   #r.PosE8 := #_w4;
   IF #_w5 THEN #Actuator.AV_Load := FALSE; END_IF;
END_REGION

REGION Network 6: Drain Inload
   RUNG wire#powerrail
      Contact( #alwaysON )
      wire#w1
      Mul(in1 := #Param.Drain_Inload_SP, in2 := 1000, out => #Drain_Inload_MSec)
   END_RUNG
   RUNG wire#w1
      Contact( #State.Inload_Enable )
      Contact( #Cmd.Drain_In )
      Coil( #State.Drain_Inload )
   END_RUNG
   RUNG wire#w1
      I_Contact( #Cmd.Inload_Select_Tank_1 )
      I_Contact( #Cmd.Inload_Select_Tank_2 )
      I_Contact( #Cmd.Inload_Select_Tank_3 )
      wire#w2
      P_Trig( #r.PosE11 )
      R_Coil( #Cmd.Drain_In )
   END_RUNG
   RUNG wire#w1
      I_Contact( #State.Inload_Enable )
   END_RUNG wire#w2
   RUNG wire#w1
      Contact( #State.Tank_inloading )
      Contact( #State.Drain_Inload )
      Contact( "AlwaysFALSE" )
      { S7_Templates := "value_type := DInt" } #Drain_Inload_Count.CTU(r := wire#w3, pv := #Param.Drain_Inload_SP, cv => #Drain_Inload_Act)
   END_RUNG
   RUNG wire#powerrail
      I_Contact( #State.Tank_inloading )
   END_RUNG wire#w3
   RUNG wire#powerrail
      I_Contact( #State.Drain_Inload )
   END_RUNG wire#w3
   // the same network as SCL:
   IF #alwaysON THEN #Drain_Inload_MSec := #Param.Drain_Inload_SP * 1000; END_IF;
   #State.Drain_Inload := #alwaysON AND #State.Inload_Enable AND #Cmd.Drain_In;
   #_w1 := #alwaysON AND ((NOT #Cmd.Inload_Select_Tank_1 AND NOT #Cmd.Inload_Select_Tank_2 AND NOT #Cmd.Inload_Select_Tank_3) OR NOT #State.Inload_Enable);
   #_w2 := #_w1 AND NOT #r.PosE11;   // rising edge
   #r.PosE11 := #_w1;
   IF #_w2 THEN #Cmd.Drain_In := FALSE; END_IF;
   #Drain_Inload_Count.CTU(CU := #alwaysON AND #State.Tank_inloading AND #State.Drain_Inload AND "AlwaysFALSE",
                           R := NOT #State.Tank_inloading OR NOT #State.Drain_Inload,
                           PV := #Param.Drain_Inload_SP,
                           CV => #Drain_Inload_Act);
END_REGION

REGION Network 7: Command Transfer to Filling
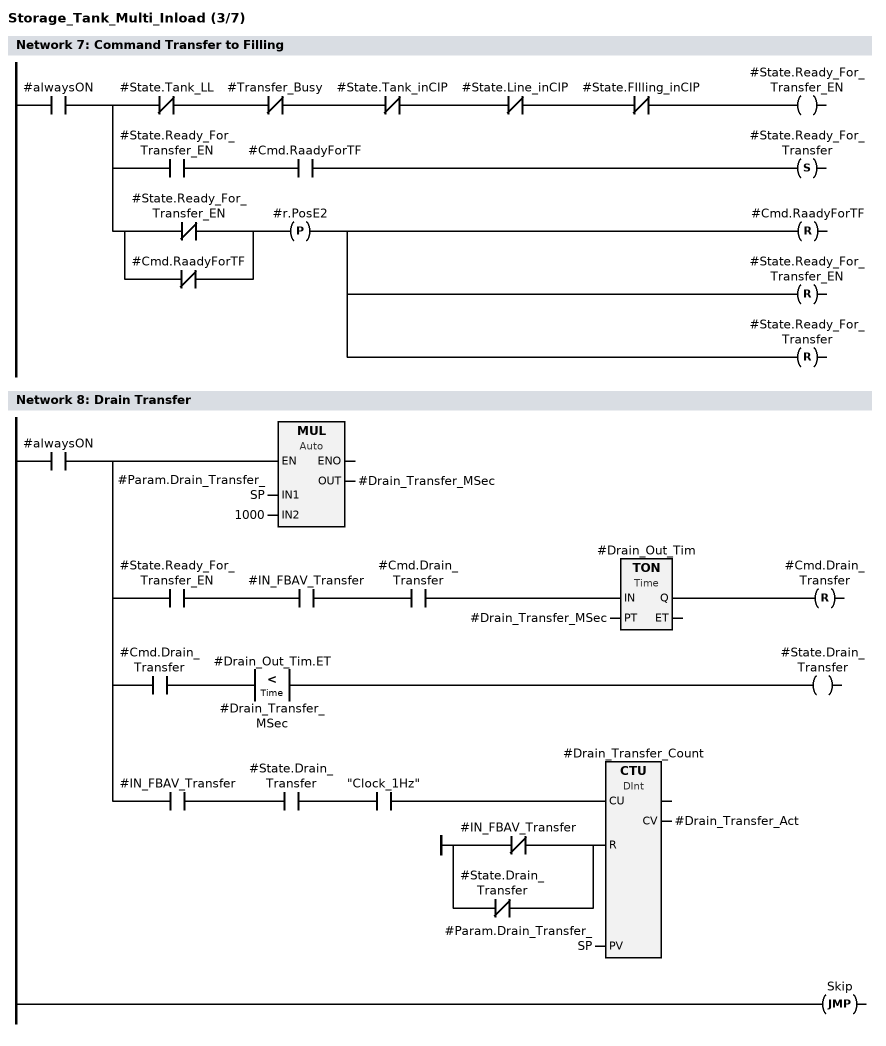
   RUNG wire#powerrail
      Contact( #alwaysON )
      wire#w1
      I_Contact( #State.Tank_LL )
      I_Contact( #Transfer_Busy )
      I_Contact( #State.Tank_inCIP )
      I_Contact( #State.Line_inCIP )
      I_Contact( #State.FIlling_inCIP )
      Coil( #State.Ready_For_Transfer_EN )
   END_RUNG
   RUNG wire#w1
      Contact( #State.Ready_For_Transfer_EN )
      Contact( #Cmd.RaadyForTF )
      S_Coil( #State.Ready_For_Transfer )
   END_RUNG
   RUNG wire#w1
      I_Contact( #State.Ready_For_Transfer_EN )
      wire#w2
      P_Trig( #r.PosE2 )
      wire#w3
      R_Coil( #Cmd.RaadyForTF )
   END_RUNG
   RUNG wire#w1
      I_Contact( #Cmd.RaadyForTF )
   END_RUNG wire#w2
   RUNG wire#w3
      R_Coil( #State.Ready_For_Transfer_EN )
   END_RUNG
   RUNG wire#w3
      R_Coil( #State.Ready_For_Transfer )
   END_RUNG
   // the same network as SCL:
   #State.Ready_For_Transfer_EN := #alwaysON AND NOT #State.Tank_LL AND NOT #Transfer_Busy AND NOT #State.Tank_inCIP AND NOT #State.Line_inCIP AND NOT #State.FIlling_inCIP;
   IF #alwaysON AND #State.Ready_For_Transfer_EN AND #Cmd.RaadyForTF THEN
       #State.Ready_For_Transfer := TRUE;
   END_IF;
   #_w1 := #alwaysON AND (NOT #State.Ready_For_Transfer_EN OR NOT #Cmd.RaadyForTF);
   #_w2 := #_w1 AND NOT #r.PosE2;   // rising edge
   #r.PosE2 := #_w1;
   IF #_w2 THEN
       #Cmd.RaadyForTF := FALSE;
       #State.Ready_For_Transfer_EN := FALSE;
       #State.Ready_For_Transfer := FALSE;
   END_IF;
END_REGION

REGION Network 8: Drain Transfer
   RUNG wire#powerrail
      Contact( #alwaysON )
      wire#w1
      Mul(in1 := #Param.Drain_Transfer_SP, in2 := 1000, out => #Drain_Transfer_MSec)
   END_RUNG
   RUNG wire#w1
      Contact( #State.Ready_For_Transfer_EN )
      Contact( #IN_FBAV_Transfer )
      Contact( #Cmd.Drain_Transfer )
      { S7_Templates := "time_type := Time" } #Drain_Out_Tim.TON(pt := #Drain_Transfer_MSec, et =>)
      R_Coil( #Cmd.Drain_Transfer )
   END_RUNG
   RUNG wire#w1
      Contact( #Cmd.Drain_Transfer )
      { S7_Templates := "SrcType := Time" } LT_Contact(in1 := #Drain_Out_Tim.ET, in2 := #Drain_Transfer_MSec)
      Coil( #State.Drain_Transfer )
   END_RUNG
   RUNG wire#w1
      Contact( #IN_FBAV_Transfer )
      Contact( #State.Drain_Transfer )
      Contact( "Clock_1Hz" )
      { S7_Templates := "value_type := DInt" } #Drain_Transfer_Count.CTU(r := wire#w2, pv := #Param.Drain_Transfer_SP, cv => #Drain_Transfer_Act)
   END_RUNG
   RUNG wire#powerrail
      I_Contact( #IN_FBAV_Transfer )
   END_RUNG wire#w2
   RUNG wire#powerrail
      I_Contact( #State.Drain_Transfer )
   END_RUNG wire#w2
   RUNG wire#powerrail
      JumpCoil( Skip )
   END_RUNG
   // the same network as SCL:
   IF #alwaysON THEN #Drain_Transfer_MSec := #Param.Drain_Transfer_SP * 1000; END_IF;
   #Drain_Out_Tim(IN := #alwaysON AND #State.Ready_For_Transfer_EN AND #IN_FBAV_Transfer AND #Cmd.Drain_Transfer,   // TON
                  PT := #Drain_Transfer_MSec);
   IF #Drain_Out_Tim.Q THEN #Cmd.Drain_Transfer := FALSE; END_IF;
   #State.Drain_Transfer := #alwaysON AND #Cmd.Drain_Transfer AND (#Drain_Out_Tim.ET < #Drain_Transfer_MSec);
   #Drain_Transfer_Count.CTU(CU := #alwaysON AND #IN_FBAV_Transfer AND #State.Drain_Transfer AND "Clock_1Hz",
                           R := NOT #IN_FBAV_Transfer OR NOT #State.Drain_Transfer,
                           PV := #Param.Drain_Transfer_SP,
                           CV => #Drain_Transfer_Act);
   GOTO Skip;
END_REGION

REGION Network 9: -----------------------------------------------State transfer to filling
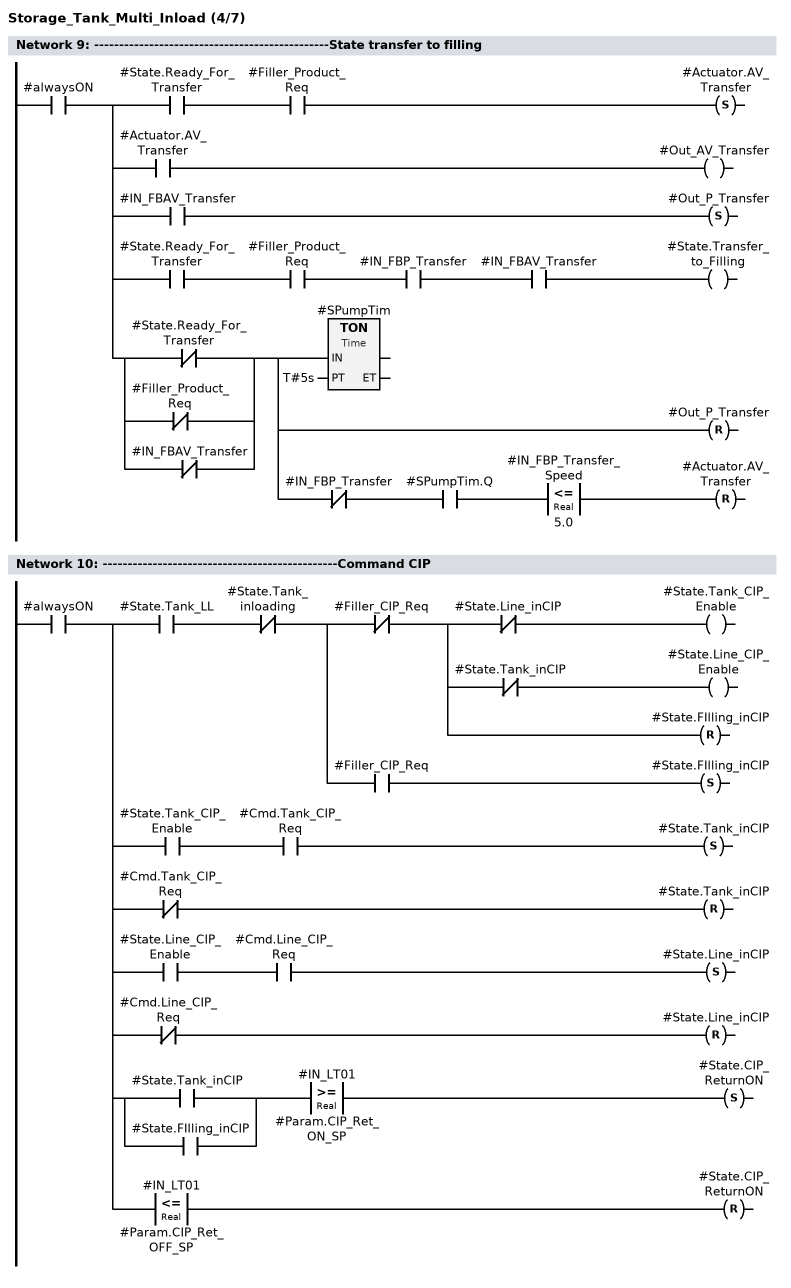
   RUNG wire#powerrail
      Contact( #alwaysON )
      wire#w1
      Contact( #State.Ready_For_Transfer )
      Contact( #Filler_Product_Req )
      S_Coil( #Actuator.AV_Transfer )
   END_RUNG
   RUNG wire#w1
      Contact( #Actuator.AV_Transfer )
      Coil( #Out_AV_Transfer )
   END_RUNG
   RUNG wire#w1
      Contact( #IN_FBAV_Transfer )
      S_Coil( #Out_P_Transfer )
   END_RUNG
   RUNG wire#w1
      Contact( #State.Ready_For_Transfer )
      Contact( #Filler_Product_Req )
      Contact( #IN_FBP_Transfer )
      Contact( #IN_FBAV_Transfer )
      Coil( #State.Transfer_to_Filling )
   END_RUNG
   RUNG wire#w1
      I_Contact( #State.Ready_For_Transfer )
      wire#w2
      { S7_Templates := "time_type := Time" } #SPumpTim.TON(pt := T#5s, et =>)
   END_RUNG
   RUNG wire#w1
      I_Contact( #Filler_Product_Req )
   END_RUNG wire#w2
   RUNG wire#w1
      I_Contact( #IN_FBAV_Transfer )
   END_RUNG wire#w2
   RUNG wire#w2
      R_Coil( #Out_P_Transfer )
   END_RUNG
   RUNG wire#w2
      I_Contact( #IN_FBP_Transfer )
      Contact( #SPumpTim.Q )
      { S7_Templates := "SrcType := Real" } LE_Contact(in1 := #IN_FBP_Transfer_Speed, in2 := 5.0)
      R_Coil( #Actuator.AV_Transfer )
   END_RUNG
   // the same network as SCL:
   IF #alwaysON AND #State.Ready_For_Transfer AND #Filler_Product_Req THEN
       #Actuator.AV_Transfer := TRUE;
   END_IF;
   #Out_AV_Transfer := #alwaysON AND #Actuator.AV_Transfer;
   IF #alwaysON AND #IN_FBAV_Transfer THEN #Out_P_Transfer := TRUE; END_IF;
   #State.Transfer_to_Filling := #alwaysON AND #State.Ready_For_Transfer AND #Filler_Product_Req AND #IN_FBP_Transfer AND #IN_FBAV_Transfer;
   #_w1 := #alwaysON AND (NOT #State.Ready_For_Transfer OR NOT #Filler_Product_Req OR NOT #IN_FBAV_Transfer);
   #SPumpTim(IN := #_w1, PT := T#5s);   // TON
   IF #_w1 THEN #Out_P_Transfer := FALSE; END_IF;
   IF #_w1 AND NOT #IN_FBP_Transfer AND #SPumpTim.Q AND (#IN_FBP_Transfer_Speed <= 5.0) THEN
       #Actuator.AV_Transfer := FALSE;
   END_IF;
END_REGION

REGION Network 10: -----------------------------------------------Command CIP
   RUNG wire#powerrail
      Contact( #alwaysON )
      wire#w1
      Contact( #State.Tank_LL )
      I_Contact( #State.Tank_inloading )
      wire#w2
      I_Contact( #Filler_CIP_Req )
      wire#w3
      I_Contact( #State.Line_inCIP )
      Coil( #State.Tank_CIP_Enable )
   END_RUNG
   RUNG wire#w3
      I_Contact( #State.Tank_inCIP )
      Coil( #State.Line_CIP_Enable )
   END_RUNG
   RUNG wire#w3
      R_Coil( #State.FIlling_inCIP )
   END_RUNG
   RUNG wire#w2
      Contact( #Filler_CIP_Req )
      S_Coil( #State.FIlling_inCIP )
   END_RUNG
   RUNG wire#w1
      Contact( #State.Tank_CIP_Enable )
      Contact( #Cmd.Tank_CIP_Req )
      S_Coil( #State.Tank_inCIP )
   END_RUNG
   RUNG wire#w1
      I_Contact( #Cmd.Tank_CIP_Req )
      R_Coil( #State.Tank_inCIP )
   END_RUNG
   RUNG wire#w1
      Contact( #State.Line_CIP_Enable )
      Contact( #Cmd.Line_CIP_Req )
      S_Coil( #State.Line_inCIP )
   END_RUNG
   RUNG wire#w1
      I_Contact( #Cmd.Line_CIP_Req )
      R_Coil( #State.Line_inCIP )
   END_RUNG
   RUNG wire#w1
      Contact( #State.Tank_inCIP )
      wire#w4
      { S7_Templates := "SrcType := Real" } GE_Contact(in1 := #IN_LT01, in2 := #Param.CIP_Ret_ON_SP)
      S_Coil( #State.CIP_ReturnON )
   END_RUNG
   RUNG wire#w1
      Contact( #State.FIlling_inCIP )
   END_RUNG wire#w4
   RUNG wire#w1
      { S7_Templates := "SrcType := Real" } LE_Contact(in1 := #IN_LT01, in2 := #Param.CIP_Ret_OFF_SP)
      R_Coil( #State.CIP_ReturnON )
   END_RUNG
   // the same network as SCL:
   #_w1 := #alwaysON AND #State.Tank_LL AND NOT #State.Tank_inloading;
   #_w2 := #_w1 AND NOT #Filler_CIP_Req;
   #State.Tank_CIP_Enable := #_w2 AND NOT #State.Line_inCIP;
   #State.Line_CIP_Enable := #_w2 AND NOT #State.Tank_inCIP;
   IF #_w2 THEN #State.FIlling_inCIP := FALSE; END_IF;
   IF #_w1 AND #Filler_CIP_Req THEN #State.FIlling_inCIP := TRUE; END_IF;
   IF #alwaysON AND #State.Tank_CIP_Enable AND #Cmd.Tank_CIP_Req THEN #State.Tank_inCIP := TRUE; END_IF;
   IF #alwaysON AND NOT #Cmd.Tank_CIP_Req THEN #State.Tank_inCIP := FALSE; END_IF;
   IF #alwaysON AND #State.Line_CIP_Enable AND #Cmd.Line_CIP_Req THEN #State.Line_inCIP := TRUE; END_IF;
   IF #alwaysON AND NOT #Cmd.Line_CIP_Req THEN #State.Line_inCIP := FALSE; END_IF;
   IF #alwaysON AND (#State.Tank_inCIP OR #State.FIlling_inCIP) AND (#IN_LT01 >= #Param.CIP_Ret_ON_SP) THEN
       #State.CIP_ReturnON := TRUE;
   END_IF;
   IF #alwaysON AND (#IN_LT01 <= #Param.CIP_Ret_OFF_SP) THEN #State.CIP_ReturnON := FALSE; END_IF;
END_REGION

REGION Network 11: Command CIP New
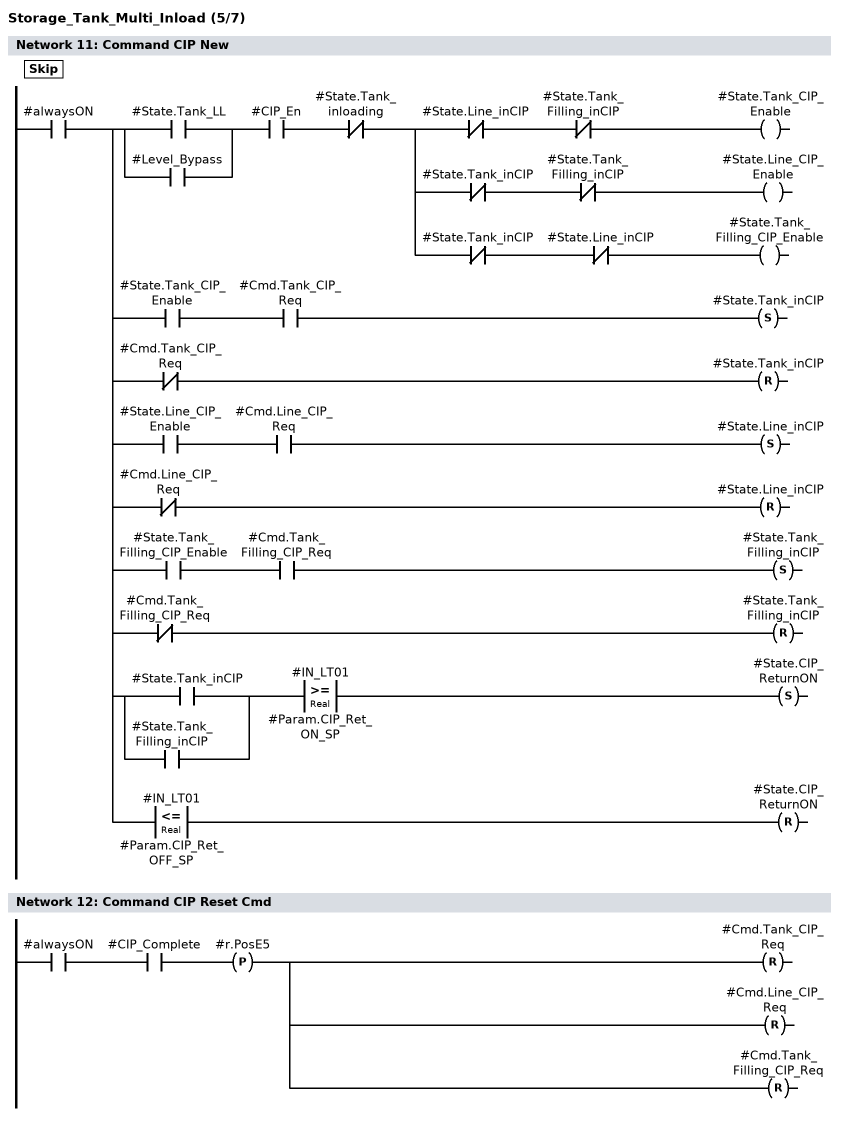
   Label( Skip )
   RUNG wire#powerrail
      Contact( #alwaysON )
      wire#w1
      Contact( #State.Tank_LL )
      wire#w2
      Contact( #CIP_En )
      I_Contact( #State.Tank_inloading )
      wire#w3
      I_Contact( #State.Line_inCIP )
      I_Contact( #State.Tank_Filling_inCIP )
      Coil( #State.Tank_CIP_Enable )
   END_RUNG
   RUNG wire#w1
      Contact( #Level_Bypass )
   END_RUNG wire#w2
   RUNG wire#w3
      I_Contact( #State.Tank_inCIP )
      I_Contact( #State.Tank_Filling_inCIP )
      Coil( #State.Line_CIP_Enable )
   END_RUNG
   RUNG wire#w3
      I_Contact( #State.Tank_inCIP )
      I_Contact( #State.Line_inCIP )
      Coil( #State.Tank_Filling_CIP_Enable )
   END_RUNG
   RUNG wire#w1
      Contact( #State.Tank_CIP_Enable )
      Contact( #Cmd.Tank_CIP_Req )
      S_Coil( #State.Tank_inCIP )
   END_RUNG
   RUNG wire#w1
      I_Contact( #Cmd.Tank_CIP_Req )
      R_Coil( #State.Tank_inCIP )
   END_RUNG
   RUNG wire#w1
      Contact( #State.Line_CIP_Enable )
      Contact( #Cmd.Line_CIP_Req )
      S_Coil( #State.Line_inCIP )
   END_RUNG
   RUNG wire#w1
      I_Contact( #Cmd.Line_CIP_Req )
      R_Coil( #State.Line_inCIP )
   END_RUNG
   RUNG wire#w1
      Contact( #State.Tank_Filling_CIP_Enable )
      Contact( #Cmd.Tank_Filling_CIP_Req )
      S_Coil( #State.Tank_Filling_inCIP )
   END_RUNG
   RUNG wire#w1
      I_Contact( #Cmd.Tank_Filling_CIP_Req )
      R_Coil( #State.Tank_Filling_inCIP )
   END_RUNG
   RUNG wire#w1
      Contact( #State.Tank_inCIP )
      wire#w4
      { S7_Templates := "SrcType := Real" } GE_Contact(in1 := #IN_LT01, in2 := #Param.CIP_Ret_ON_SP)
      S_Coil( #State.CIP_ReturnON )
   END_RUNG
   RUNG wire#w1
      Contact( #State.Tank_Filling_inCIP )
   END_RUNG wire#w4
   RUNG wire#w1
      { S7_Templates := "SrcType := Real" } LE_Contact(in1 := #IN_LT01, in2 := #Param.CIP_Ret_OFF_SP)
      R_Coil( #State.CIP_ReturnON )
   END_RUNG
   // the same network as SCL:
   Skip:
   #_w1 := #alwaysON AND (#State.Tank_LL OR #Level_Bypass) AND #CIP_En AND NOT #State.Tank_inloading;
   #State.Tank_CIP_Enable := #_w1 AND NOT #State.Line_inCIP AND NOT #State.Tank_Filling_inCIP;
   #State.Line_CIP_Enable := #_w1 AND NOT #State.Tank_inCIP AND NOT #State.Tank_Filling_inCIP;
   #State.Tank_Filling_CIP_Enable := #_w1 AND NOT #State.Tank_inCIP AND NOT #State.Line_inCIP;
   IF #alwaysON AND #State.Tank_CIP_Enable AND #Cmd.Tank_CIP_Req THEN #State.Tank_inCIP := TRUE; END_IF;
   IF #alwaysON AND NOT #Cmd.Tank_CIP_Req THEN #State.Tank_inCIP := FALSE; END_IF;
   IF #alwaysON AND #State.Line_CIP_Enable AND #Cmd.Line_CIP_Req THEN #State.Line_inCIP := TRUE; END_IF;
   IF #alwaysON AND NOT #Cmd.Line_CIP_Req THEN #State.Line_inCIP := FALSE; END_IF;
   IF #alwaysON AND #State.Tank_Filling_CIP_Enable AND #Cmd.Tank_Filling_CIP_Req THEN
       #State.Tank_Filling_inCIP := TRUE;
   END_IF;
   IF #alwaysON AND NOT #Cmd.Tank_Filling_CIP_Req THEN #State.Tank_Filling_inCIP := FALSE; END_IF;
   IF #alwaysON AND (#State.Tank_inCIP OR #State.Tank_Filling_inCIP) AND (#IN_LT01 >= #Param.CIP_Ret_ON_SP) THEN
       #State.CIP_ReturnON := TRUE;
   END_IF;
   IF #alwaysON AND (#IN_LT01 <= #Param.CIP_Ret_OFF_SP) THEN #State.CIP_ReturnON := FALSE; END_IF;
END_REGION

REGION Network 12: Command CIP Reset Cmd
   RUNG wire#powerrail
      Contact( #alwaysON )
      Contact( #CIP_Complete )
      P_Trig( #r.PosE5 )
      wire#w1
      R_Coil( #Cmd.Tank_CIP_Req )
   END_RUNG
   RUNG wire#w1
      R_Coil( #Cmd.Line_CIP_Req )
   END_RUNG
   RUNG wire#w1
      R_Coil( #Cmd.Tank_Filling_CIP_Req )
   END_RUNG
   // the same network as SCL:
   #_w1 := #alwaysON AND #CIP_Complete;
   #_w2 := #_w1 AND NOT #r.PosE5;   // rising edge
   #r.PosE5 := #_w1;
   IF #_w2 THEN
       #Cmd.Tank_CIP_Req := FALSE;
       #Cmd.Line_CIP_Req := FALSE;
       #Cmd.Tank_Filling_CIP_Req := FALSE;
   END_IF;
END_REGION

REGION Network 13: Send CIP Request
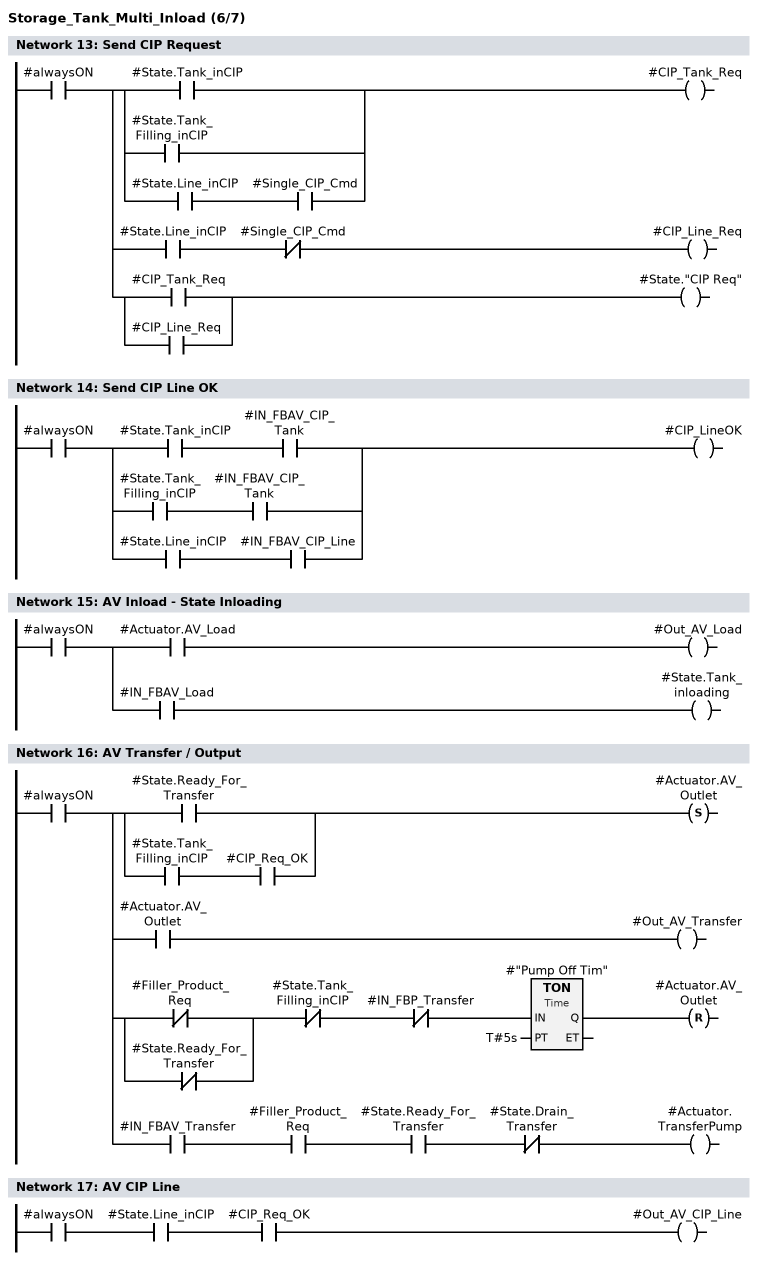
   RUNG wire#powerrail
      Contact( #alwaysON )
      wire#w1
      Contact( #State.Tank_inCIP )
      wire#w2
      Coil( #CIP_Tank_Req )
   END_RUNG
   RUNG wire#w1
      Contact( #State.Tank_Filling_inCIP )
   END_RUNG wire#w2
   RUNG wire#w1
      Contact( #State.Line_inCIP )
      Contact( #Single_CIP_Cmd )
   END_RUNG wire#w2
   RUNG wire#w1
      Contact( #State.Line_inCIP )
      I_Contact( #Single_CIP_Cmd )
      Coil( #CIP_Line_Req )
   END_RUNG
   RUNG wire#w1
      Contact( #CIP_Tank_Req )
      wire#w3
      Coil( #State."CIP Req" )
   END_RUNG
   RUNG wire#w1
      Contact( #CIP_Line_Req )
   END_RUNG wire#w3
   // the same network as SCL:
   #CIP_Tank_Req := #alwaysON AND (#State.Tank_inCIP OR #State.Tank_Filling_inCIP OR (#State.Line_inCIP AND #Single_CIP_Cmd));
   #CIP_Line_Req := #alwaysON AND #State.Line_inCIP AND NOT #Single_CIP_Cmd;
   #State."CIP Req" := #alwaysON AND (#CIP_Tank_Req OR #CIP_Line_Req);
END_REGION

REGION Network 14: Send CIP Line OK
   RUNG wire#powerrail
      Contact( #alwaysON )
      wire#w1
      Contact( #State.Tank_inCIP )
      Contact( #IN_FBAV_CIP_Tank )
      wire#w2
      Coil( #CIP_LineOK )
   END_RUNG
   RUNG wire#w1
      Contact( #State.Tank_Filling_inCIP )
      Contact( #IN_FBAV_CIP_Tank )
   END_RUNG wire#w2
   RUNG wire#w1
      Contact( #State.Line_inCIP )
      Contact( #IN_FBAV_CIP_Line )
   END_RUNG wire#w2
   // the same network as SCL:
   #CIP_LineOK := #alwaysON AND ((#State.Tank_inCIP AND #IN_FBAV_CIP_Tank) OR (#State.Tank_Filling_inCIP AND #IN_FBAV_CIP_Tank) OR (#State.Line_inCIP AND #IN_FBAV_CIP_Line));
END_REGION

REGION Network 15: AV Inload - State Inloading
   RUNG wire#powerrail
      Contact( #alwaysON )
      wire#w1
      Contact( #Actuator.AV_Load )
      Coil( #Out_AV_Load )
   END_RUNG
   RUNG wire#w1
      Contact( #IN_FBAV_Load )
      Coil( #State.Tank_inloading )
   END_RUNG
   // the same network as SCL:
   #Out_AV_Load := #alwaysON AND #Actuator.AV_Load;
   #State.Tank_inloading := #alwaysON AND #IN_FBAV_Load;
END_REGION

REGION Network 16: AV Transfer / Output
   RUNG wire#powerrail
      Contact( #alwaysON )
      wire#w1
      Contact( #State.Ready_For_Transfer )
      wire#w2
      S_Coil( #Actuator.AV_Outlet )
   END_RUNG
   RUNG wire#w1
      Contact( #State.Tank_Filling_inCIP )
      Contact( #CIP_Req_OK )
   END_RUNG wire#w2
   RUNG wire#w1
      Contact( #Actuator.AV_Outlet )
      Coil( #Out_AV_Transfer )
   END_RUNG
   RUNG wire#w1
      I_Contact( #Filler_Product_Req )
      wire#w3
      I_Contact( #State.Tank_Filling_inCIP )
      I_Contact( #IN_FBP_Transfer )
      { S7_Templates := "time_type := Time" } #"Pump Off Tim".TON(pt := T#5s, et =>)
      R_Coil( #Actuator.AV_Outlet )
   END_RUNG
   RUNG wire#w1
      I_Contact( #State.Ready_For_Transfer )
   END_RUNG wire#w3
   RUNG wire#w1
      Contact( #IN_FBAV_Transfer )
      Contact( #Filler_Product_Req )
      Contact( #State.Ready_For_Transfer )
      I_Contact( #State.Drain_Transfer )
      Coil( #Actuator.TransferPump )
   END_RUNG
   // the same network as SCL:
   IF #alwaysON AND (#State.Ready_For_Transfer OR (#State.Tank_Filling_inCIP AND #CIP_Req_OK)) THEN
       #Actuator.AV_Outlet := TRUE;
   END_IF;
   #Out_AV_Transfer := #alwaysON AND #Actuator.AV_Outlet;
   #"Pump Off Tim"(IN := #alwaysON AND (NOT #Filler_Product_Req OR NOT #State.Ready_For_Transfer) AND NOT #State.Tank_Filling_inCIP AND NOT #IN_FBP_Transfer,   // TON
                   PT := T#5s);
   IF #"Pump Off Tim".Q THEN #Actuator.AV_Outlet := FALSE; END_IF;
   #Actuator.TransferPump := #alwaysON AND #IN_FBAV_Transfer AND #Filler_Product_Req AND #State.Ready_For_Transfer AND NOT #State.Drain_Transfer;
END_REGION

REGION Network 17: AV CIP Line
   RUNG wire#powerrail
      Contact( #alwaysON )
      Contact( #State.Line_inCIP )
      Contact( #CIP_Req_OK )
      Coil( #Out_AV_CIP_Line )
   END_RUNG
   // the same network as SCL:
   #Out_AV_CIP_Line := #alwaysON AND #State.Line_inCIP AND #CIP_Req_OK;
END_REGION

REGION Network 18: AV CIP Tank to Filling
